this function calculates the polynom C[0] + C[1]*X^1 + C[2]*X^2 * C[3]*X^3 + C[4]*X^4 + C[5]*X^5 + C[6]*X^6 + C[7]*X^7

*)

F_POLY := ((((((( c[7] * x + c[6] ) * x + c[5] ) * x + c[4] ) * x + c[3] ) * x + c[2] ) * x + c[1] ) * x + c[0] ) ;


(* revision history
hm		20. may. 2008		rev 1.0
	original version

hm	18. mar. 2011	rev 1.1
	improved performance
*)

END_FUNCTION

// POUs/Mathematical/functions/F_POWER
FUNCTION F_POWER : REAL
VAR_INPUT
	a : REAL;
	x : REAL;
	n : REAL;
END_VAR


(*
version 1.0	1 sep 2006
programmer 	hugo
tested by		tobias

this function calculates the power equation f_power = a*x^n

*)

F_POWER := a * EXPT(X, N);

END_FUNCTION

// POUs/Mathematical/functions/F_QUAD
FUNCTION F_QUAD : REAL
VAR_INPUT
	X : REAL;
	A : REAL;
	B : REAL;
	C : REAL;
END_VAR


(*
version 1.1	18. Mar. 2011
programmer 	hugo
tested by		tobias

this function calculates the quadratic equation f_lin = a*x + b

*)

F_QUAD :=  (A * X + B) * X + C;

(* revision history

hm	1. sep. 2006	rev 1.0
	original version

hm	18. mar. 2001	rev 1.1
	improved performance
*)

END_FUNCTION

// POUs/Engineering/conversion/F_TO_C
FUNCTION F_TO_C : REAL
VAR_INPUT
	fahrenheit : REAL;
END_VAR


(*
version 1.1	11. mar. 2009
programmer 	hugo
tested BY		tobias

this FUNCTION converts fahrenheit TO celsius

*)

F_TO_C := (fahrenheit - 32.0) * 0.5555555555555;

(* revision history
hm	4. aug 2006	rev 1.0
	original version

hm	11. mar. 2009	rev 1.1
	real constants updated to new systax using dot

*)

END_FUNCTION

// POUs/Engineering/conversion/F_TO_OM
FUNCTION F_TO_OM : REAL
VAR_INPUT
	F : REAL;
END_VAR


(*
version 1.1	18. oct. 2008
programmer 	hugo
tested by	oscat

this function converts frequency to Omega F
Omega = 2*PI*F
*)

F_TO_OM := math.PI2 * F;


(* revision history
hm	22. jan. 2007	rev 1.0
	original version

hm	18. oct. 2008	rev 1.1
	unsing math constants

*)

END_FUNCTION

// POUs/Engineering/conversion/F_TO_PT
FUNCTION F_TO_PT : TIME
VAR_INPUT
	F : REAL;
END_VAR


(*
version 1.1	11. mar. 2009
programmer 	hugo
tested by		tobias

this function converts frequency to periode time  
*)

F_TO_PT := DWORD_TO_TIME(REAL_TO_DWORD(1.0 / F * 1000.0));


(* revision history

hm	4. aug. 2006	rev 1.0
	original version

hm	11. mar. 2009	rev 1.1
	real constants updated to new systax using dot

*)

END_FUNCTION

// POUs/Mathematical/FACT
FUNCTION FACT : DINT
VAR_INPUT
	X : INT;
END_VAR


(*
version 1.5	26. mar. 2011
programmer 	hugo
tested by		tobias

this function calculates the factorial of x

if the input is negative or higher then 12 the output will be -1.

*)

IF X >= 0 AND X <= 12 THEN
	FACT := math.FACTS[X];
ELSE
	FACT := -1;
END_IF;


(* working code without array
IF X > 12 OR X < 0 THEN
	FACT := -1;
ELSIF X < 7 THEN
	FACT := 1;
	FOR i := 2 TO X DO
		FACT := FACT * i;
	END_FOR;
ELSE
	FACT := 5040;
	FOR i := 8 TO X DO
		FACT := FACT * i;
	END_FOR;
END_IF;
*)

(* revision history
hm 4.3.2007		rev 1.1
	changed a critical error where while loop was indefinite.

hm	10.12.2007	rev 1.2
	start value for i has changed to 2 for better performance

hm	10. mar 2008	rev 1.3
	changed output of fact to dint to allow bigger values

hm	27. oct. 2008	rev 1.4
	optimized code

hm	26. mar. 2011	rev 1.5
	using array math.facts
*)

END_FUNCTION

// POUs/Engineering/signal processing/FADE
FUNCTION_BLOCK FADE
VAR_INPUT
	IN1 : REAL;
	IN2 : REAL;
	F : BOOL;
	TF : TIME;
	rst : BOOL;
END_VAR
VAR_OUTPUT
	Y : REAL;
END_VAR
VAR
	rmx : RMP_W;
END_VAR

(*
version 1.3	24. jan. 2009
programmer 	oscat
tested BY		oscat

FADE is used to crossfade between the inputs IN1 and IN2. The fade_over time is specified with TF.
When F = TRUE then Y = IN2 after the time TF, and when F = FALSE then Y = IN1.

*)

rmx(rst := rst AND NOT F, set := rst AND F, pt := TF, up := F);
Y := (in2 - In1) / 65535.0 * WORD_TO_REAL(rmx.out) + in1;


(* code for rev 1.1
IF rst THEN
	rmx(set := F, rst := NOT F);
ELSIF F AND (NOT rmx.high) THEN
	rmx(PT := TF, UP := TRUE, e := TRUE, rst := FALSE, set := FALSE);
ELSIF (NOT F) AND (NOT rmx.low) THEN
	rmx(PT := TF, UP := FALSE, e := TRUE, rst := FALSE, set := FALSE);
ELSE
	rmx(e := FALSE, rst := FALSE, set := FALSE);
END_IF;
Y := (WORD_TO_REAL(rmx.out) * in1 + WORD_TO_REAL(FF - rmx.out) * IN2) / FF;
*)


(* revision history
hm	26. dec 2007	rev 1.0
	original version

hm	18. oct. 2008	rev 1.1
	improved performance
	changed calls for rmp_w because rmp_w has chaged

hm	17. dec. 2008	rev 1.2
	function of input f was inverted

hm	24. jan. 2009	rev 1.3
	delted unused var FF
*)

END_FUNCTION_BLOCK

// POUs/Engineering/signal generators/RMP_W
FUNCTION_BLOCK RMP_W
VAR_INPUT
	SET : BOOL;
	PT : TIME;
	E : BOOL := TRUE;
	UP : BOOL := TRUE;
	RST : BOOL;
END_VAR
VAR_OUTPUT
	out : WORD;
	busy : BOOL;
	high : BOOL;
	low : BOOL;
END_VAR
VAR
	rmp : _RMP_W;
END_VAR

(*
version 2.0	23. oct. 2008
programmer 	oscat
tested BY	oscat

this ramp generator generates a Word wide ramp with 65535 steps
the generator has an asynchronous set and reset
the ramp is controlled by PT which is the total ramp time for a full sweep from 0..65535
an UD input controlls the direction Up or Down and the E input enables the ramp generation
a busy output indicates that the ramp is running, busy false means output is stable.
the outputs low and high will be true when the output has reached its max or min value.
*)

(* generate ramp *)
rmp(dir := UP, E := E, TR := PT, rmp := out);

(* set or reset operation *)
IF RST THEN
	out := 0;
ELSIF SET THEN
	out := 65535;
END_IF;

(* checks for outputs stable and reset or set busy flag *)
low := out = 0;
high := out = 65535;
busy := NOT (low OR high) AND E;


(* revision history:

hm 4.10.2006		rev 1.1
	added the busy output which signals that the ramp is running.

hm 22.1.2007		rev 1.2
	deleted unused variable step

hm	17.9.2007		rev 1.3
	replaced time() with t_plc_ms() for compatibility reasons

hm	28. sep 2007	rev 1.4
	added outputs on and off
	busy is now disabled while en is false
	new coding for higher accuracy and performance

hm	5. oct 2007	rev 1.5
	added statements to allow for PT to be t#0s output jumps to max or min immediately

hm	2. dec 2007	rev 1.6
	corrected an error in calculation of step response

hm	25. dec 2007	rev 1.7
	corrected an error while step response was too slow for fast rise times

hm	16. oct. 2008	rev 1.8
	improved performance

hm	18. oct. 2008	rev 1.9
	renamed inout EN to E for compatibility reasons

hm	23. oct. 2008	rev 2.0
	new code using _RMP_W
*)

END_FUNCTION_BLOCK

// POUs/Logic/FF edge triggered/FF_D2E
FUNCTION_BLOCK FF_D2E
VAR_INPUT
	D0 : BOOL;
	D1 : BOOL;
	CLK : BOOL;
	RST : BOOL;
END_VAR
VAR_OUTPUT
	Q0 : BOOL;
	Q1 : BOOL;
END_VAR
VAR
	edge : BOOL;
END_VAR

(*
version 1.3	14. mar. 2009
programmer 	hugo
tested by		oscat

dual D-type flip flop with reset and rising clock trigger

*)

IF rst THEN
	Q0 := FALSE;
	Q1 := FALSE;
ELSIF clk AND NOT edge THEN
	Q0 := D0;
	Q1 := D1;
END_IF;
edge := CLK;

(* revision history
hm	25. dec 2007	rev 1.0
	original version

hm	27. dec 2007	rev 1.1
	changed code for better performance

hm	30. oct. 200	rev 1.2
	deleted unnecessary init with 0

hm	14. mar. 2009	rev 1.3
	removed double assignments

*)

END_FUNCTION_BLOCK

// POUs/Logic/FF edge triggered/FF_D4E
FUNCTION_BLOCK FF_D4E
VAR_INPUT
	D0 : BOOL;
	D1 : BOOL;
	D2 : BOOL;
	D3 : BOOL;
	CLK : BOOL;
	RST : BOOL;
END_VAR
VAR_OUTPUT
	Q0 : BOOL;
	Q1 : BOOL;
	Q2 : BOOL;
	Q3 : BOOL;
END_VAR
VAR
	edge : BOOL;
END_VAR


(*
version 1.3	14. mar. 2009
programmer 	hugo
tested by		oscat

quad D-type flip flop with reset and rising clock trigger

*)

IF rst THEN
	Q0 := FALSE;
	Q1 := FALSE;
	Q2 := FALSE;
	Q3 := FALSE;
ELSIF clk AND NOT edge THEN
	Q0 := D0;
	Q1 := D1;
	Q2 := D2;
	Q3 := D3;
END_IF;
edge := CLK;

(* revision history
hm	4. aug 2006	rev 1.0
	original version

hm	27. dec 2007	rev 1.1
	changed code for better performance

hm	30. oct. 200	rev 1.2
	deleted unnecessary init with 0

hm	14. mar. 2009	rev 1.3
	removed double assignments

*)

END_FUNCTION_BLOCK

// POUs/Logic/FF edge triggered/FF_DRE
FUNCTION_BLOCK FF_DRE
VAR_INPUT
	SET : BOOL;
	D : BOOL;
	CLK : BOOL;
	RST : BOOL;
END_VAR
VAR_OUTPUT
	Q : BOOL;
END_VAR
VAR
	edge : BOOL;
END_VAR


(*
version 1.2	30. oct. 2008
programmer 	hugo
tested by	oscat

D-type flip flop with set, reset and rising clock trigger

*)

IF rst OR set THEN
	Q := NOT rst;
ELSIF clk AND NOT edge THEN
	Q := D;
END_IF;
edge := CLK;

(* revision history
hm	4. aug 2006		rev 1.0
	original version

hm	27. dec 2007	rev 1.1
	changed code for better performance

hm	30. oct. 2008	rev 1.2
	optimized performance
*)

END_FUNCTION_BLOCK

// POUs/Logic/FF edge triggered/FF_JKE
FUNCTION_BLOCK FF_JKE
VAR_INPUT
	SET : BOOL;
	J : BOOL;
	CLK : BOOL;
	K : BOOL;
	RST : BOOL;
END_VAR
VAR_OUTPUT
	Q : BOOL;
END_VAR
VAR
	edge : BOOL;
END_VAR


(*
version 1.2	30. oct. 2008
programmer 	hugo
tested by	oscat

JK-type flip flop with set, reset and rising clock trigger
set and reset are asynchron while the FF is rising edge triggered
J=0 and K=0 and CLK >>> no action
J=1 and K=0 and CLK >>> output = 1
J=0 and K=1 and CLK >>> output = 0
J=1 and K=1 and CLK >>> toggle output


*)

IF rst OR set THEN
	Q := NOT rst;
ELSIF clk AND NOT edge THEN
	IF J XOR K THEN Q := J;
	ELSE Q := K XOR Q;
	END_IF;
END_IF;
edge := CLK;

(* revision history
hm	4. aug 2006		rev 1.0
	original version

hm	27. dec 2007	rev 1.1
	changed code for better performance

hm	30. oct. 2008	rev 1.2
	optimized performance
*)

END_FUNCTION_BLOCK

// POUs/Logic/FF edge triggered/FF_RSE
FUNCTION_BLOCK FF_RSE
VAR_INPUT
	CS : BOOL;
	CR : BOOL;
	RST : BOOL;
END_VAR
VAR_OUTPUT
	Q : BOOL;
END_VAR
VAR
	es, er : BOOL;
END_VAR

(*
version 1.0	16. jul. 2008
programmer 	hugo
tested by	oscat

this is a rising edge triggered rs flip flop
a rising edge on CS sets Q = TRUE and a rising edge on CR sets Q = FALSE.
CR has priority over CS.

*)

IF rst THEN
	(* asynchronous reset *)
	Q := FALSE;
ELSIF CR AND NOT er THEN
	(* rising edge on CR *)
	Q := FALSE;
ELSIF CS AND NOT es THEN
	(* rising edge on CS *)
	Q := TRUE;
END_IF;

es := CS;
er := CR;

(* revision history

hm	16. jul. 2008	rev 1.0
	original version

*)

END_FUNCTION_BLOCK

// POUs/Mathematical/FIB
FUNCTION FIB : DINT
VAR_INPUT
	X : INT;
END_VAR
VAR
	t1, t2: DINT;
END_VAR

(*
version 1.3	26. mar. 2008
programmer 	hugo
tested by		tobias

this function calculates the fibonacci sequence

*)

IF X < 0 OR X > 46 THEN
	FIB := -1;
ELSIF x < 2 THEN
	FIB := X;
	RETURN;
ELSE
	(* the fibonacci number is the sum of the two suceeding fibonaci numbers *)
	(* we store the numbers alternatively in t1 and t2 depending on pt *)
	t2 := 1;
	WHILE X > 3 DO
		X := X-2;
		t1 := t1 + t2;
		t2 := t1 + t2;
	END_WHILE;
	IF X > 2 THEN t1 := t1 + t2; END_IF;
	fib := t1 + t2;
END_IF;

(* alternative code for very big numbers

IF X < 31 THEN
	fib := 0.4472136 * (expn(1.618034,X) - expn(-0.618034,X));
ELSE
	fib := 0.4472133 * expn(1.618034,X);
END_IF;

*)

(* revision history
hm		27. dec 2007	rev 1.0
	original version

hm		2. jan 2008	rev 1.1
	deleted unused variable pt

hm		10. mar 2008	rev 1.2
	changed output to dint instead of real

hm		26. mar. 2008	rev 1.3
	function now returns -1 for input < 0 or > 46

*)

END_FUNCTION

// POUs/Logic/memory/FIFO_16
FUNCTION_BLOCK FIFO_16
VAR_INPUT
	Din : DWORD;
	E : BOOL := TRUE;
	RD : BOOL;
	WD : BOOL;
	RST : BOOL;
END_VAR
VAR_OUTPUT
	Dout : DWORD;
	EMPTY : BOOL := TRUE;
	FULL : BOOL;
END_VAR
VAR
	fifo : ARRAY[0..n] OF DWORD;
	pr : INT;
	pw : INT;
END_VAR
VAR CONSTANT
	n : INT := 16;	(* changing this value will chage the number of stored elements in the fifo *)
END_VAR


(*
version 2.0	24. jul. 2009
programmer 	hugo
tested by		oscat

16 Dword FIFO memory
*)

IF RST THEN
	pw := pr;
	FULL := FALSE;
	EMPTY := TRUE;
	Dout := 0;
ELSIF E THEN
	IF NOT EMPTY AND RD THEN
		Dout := fifo[pr];
		pr := INC1(pr,n);
		EMPTY := pr = pw;
		FULL := FALSE;
	END_IF;
	IF NOT FULL AND WD THEN
		fifo[pw] := Din;
		pw := INC1(pw,n);
		FULL := pw = pr;
		EMPTY := FALSE;
	END_IF;
END_IF;


(* revision history

hm	4. aug. 2006	rev 1.0
	original version

hm	19. feb 2008	rev 1.1
	performance improvements

hm	17. oct. 2008	rev 1.2
	improved performance

ks	27. oct. 2008	rev 1.3
	optimized coding

hm	14. mar. 2009	rev 1.4
	removed double assignments

hm 24. jul. 2009	rev 2.0
	chaged inputs E and WR to E, WD and WR
	allow read and write in one cycle

*)

END_FUNCTION_BLOCK

// POUs/Logic/memory/FIFO_32
FUNCTION_BLOCK FIFO_32
VAR_INPUT
	Din : DWORD;
	E : BOOL := TRUE;
	RD : BOOL;
	WD : BOOL;
	RST : BOOL;
END_VAR
VAR_OUTPUT
	Dout : DWORD;
	EMPTY : BOOL := TRUE;
	FULL : BOOL;
END_VAR
VAR
	fifo : ARRAY[0..n] OF DWORD;
	pr : INT;
	pw : INT;
END_VAR
VAR CONSTANT
	n : INT := 32;	(* changing this value will chage the number of stored elements in the fifo *)
END_VAR

(*
version 2.0	24. jul. 2009
programmer 	hugo
tested by		oscat

32 Dword FIFO memory
*)

IF RST THEN
	pw := pr;
	FULL := FALSE;
	EMPTY := TRUE;
	Dout := 0;
ELSIF E THEN
	IF NOT EMPTY AND RD THEN
		Dout := fifo[pr];
		pr := INC1(pr,n);
		EMPTY := pr = pw;
		FULL := FALSE;
	END_IF;
	IF NOT FULL AND WD THEN
		fifo[pw] := Din;
		pw := INC1(pw,n);
		FULL := pw = pr;
		EMPTY := FALSE;
	END_IF;
END_IF;

(* revision history
hm	4. aug. 2006	rev 1.0
	original version

hm	19. feb 2008	rev 1.1
	performance improvements

hm	17. oct. 2008	rev 1.2
	improved performance

ks	27. oct. 2008 rev 1.3
	improved code

hm	14. mar. 2009	rev 1.4
	removed double assignments

hm 24. jul. 2009	rev 2.0
	chaged inputs E and WR to E, WD and WR
	allow read and write in one cycle

*)

END_FUNCTION_BLOCK

// POUs/Engineering/signal processing/FILTER_DW
FUNCTION_BLOCK FILTER_DW
VAR_INPUT
	X : DWORD;
	T : TIME;
END_VAR
VAR_OUTPUT
	Y : DWORD;
END_VAR
VAR
	last : DWORD;
	tx: DWORD;
	init: BOOL;
	Yi : REAL;
END_VAR

(*
version 1.1	3. nov. 2008
programmer 	hugo
tested by		oscat

FILTER_DW is an low pass filter with a programmable time T used for DWORD format.
 
*)

(* read system time *)
tx := T_PLC_MS();

(* startup initialisation *)
IF NOT init OR T = t#0s THEN
	init := TRUE;
	Yi := DWORD_TO_REAL(X);
ELSE
	Yi := Yi + (DWORD_TO_REAL(X) - DWORD_TO_REAL(Y)) * DWORD_TO_REAL(tx - last) / TIME_TO_REAL(T);
END_IF;
last := tx;

Y := REAL_TO_DWORD(Yi);



(*
hm 10. oct. 2008	rev 1.0
	original version

hm	3. nov. 2008	REV 1.1
	corrected an overflow problem
*)

END_FUNCTION_BLOCK

// POUs/Engineering/signal processing/FILTER_I
FUNCTION_BLOCK FILTER_I
VAR_INPUT
	X : INT;
	T : TIME;
END_VAR
VAR_OUTPUT
	Y : INT;
END_VAR
VAR
	Yi : DINT;
	last : DWORD;
	tx: DWORD;
	init: BOOL;
END_VAR

(*
version 1.0	8. nov. 2008
programmer 	hugo
tested by	oscat

FILTER_I is a low pass filter with a programmable time T used for INT format.
 
*)

(* read system time *)
tx := T_PLC_MS();

(* startup initialisation *)
IF NOT init OR T = t#0s THEN
	init := TRUE;
	Yi := INT_TO_DINT(X) * 1000;
ELSE
	(* to increase accuracy of the filter we calculate internal Yi wich is Y * 1000 *)
	Yi := Yi + INT_TO_DINT(X - Y) * DWORD_TO_DINT(tx - last) * 1000 / TIME_TO_DINT(T);
END_IF;
last := tx;
Y := DINT_TO_INT(yi / 1000);



(*
hm 8. nov. 2008	rev 1.0
	original version

*)

END_FUNCTION_BLOCK

// POUs/Engineering/signal processing/FILTER_MAV_DW
FUNCTION_BLOCK FILTER_MAV_DW
VAR_INPUT
	X : DWORD;
	N : UINT;
	RST : BOOL;
END_VAR
VAR_OUTPUT
	Y : DWORD;
END_VAR
VAR
	init: BOOL;
	buffer : ARRAY[0..31] OF DWORD;
	i: INT;
END_VAR
VAR_TEMP
	tmp: INT;
END_VAR

(*
version 1.3	23. feb. 2009
programmer 	hugo
tested by		oscat

FILTER_MAV_DW is a moving average filter with programmable length N for DWORD Data.
 
*)

(* limit N to size of buffer *)
N := MIN(N, 32);

(* startup initialisation *)
IF NOT init OR rst OR N = 0 THEN
	init := TRUE;
	tmp := UINT_TO_INT(N)-1;
	FOR i := 0 TO tmp DO
		buffer[i] := X;
	END_FOR;
	Y := X;
ELSE
	tmp := UINT_TO_INT(N);
	i := INC1(i, tmp);
	Y := Y + (X - buffer[i]) / N;
	buffer[i] := X;
END_IF;




(*
hm 13. oct. 2008	rev 1.0
	original version

hm	27. oct. 2008	rev 1.1
	added typecast to avoid warnings

hm	24. nov. 2008	rev 1.2
	added typecasts to avoid warnings
	avoid divide by 0 if N = 0

hm	23. feb. 2009	rev 1.3
	limit N to max array size

*)

END_FUNCTION_BLOCK

// POUs/Engineering/signal processing/FILTER_MAV_W
FUNCTION_BLOCK FILTER_MAV_W
VAR_INPUT
	X : WORD;
	N : UINT;
	RST : BOOL;
END_VAR
VAR_OUTPUT
	Y : WORD;
END_VAR
VAR
	init: BOOL;
	buffer : ARRAY[1..32] OF WORD;
	i: INT;
	sum : DWORD;
END_VAR
VAR_TEMP
	tmp : INT;
END_VAR

(*
version 1.4	26. MAR. 2011
programmer 	hugo
tested by		oscat

FILTER_MAV_W is a moving average filter with programmable length N for WORD Data.
 
*)

(* limit N to size of buffer *)
N := MIN(N, 32);

(* startup initialisation *)
IF NOT init OR rst OR N = 0 THEN
	init := TRUE;
	tmp := UINT_TO_INT(N) - 1;
	FOR i := 1 TO tmp DO
		buffer[i] := X;
	END_FOR;
	sum := Y * N;
	Y := X;
ELSE
	tmp := UINT_TO_INT(N);
	i := INC1(i, tmp);
	sum := sum + X - buffer[i];
	Y := DWORD_TO_WORD(sum / N);
	buffer[i] := X;
END_IF;



(*
hm 13. oct. 2008	rev 1.0
	original version

hm	18. oct. 2008	rev 1.1
	added typecast to avoid warnings

hm	24. nov. 2008	rev 1.2
	added typecasts to avoid warnings
	avoid devide by 0 if N = 0

hm	23. feb. 2009	rev 1.3
	limit N to max array size

hm	26. mar. 2011	rev 1.4
	corrected error in calculation
*)

END_FUNCTION_BLOCK

// POUs/Engineering/signal processing/FILTER_W
FUNCTION_BLOCK FILTER_W
VAR_INPUT
	X : WORD;
	T : TIME;
END_VAR
VAR_OUTPUT
	Y : WORD;
END_VAR
VAR
	last : DWORD;
	tx: DWORD;
	init: BOOL;
	tmp: DWORD;
END_VAR

(*
version 1.2	25. jan. 2011
programmer 	hugo
tested by	oscat

FILTER_W is an low pass filter with a programmable time T used for WORD format.
 
*)

(* read system time *)
tx := T_PLC_MS();

(* startup initialisation *)
IF NOT init OR T = T#0s THEN
	init := TRUE;
	last := tx;
	Y := X;
ELSIF Y = X THEN
	last := tx;
ELSE
	tmp :=  WORD_TO_DWORD(X - Y) * (tx - last) / TIME_TO_DWORD(T);
	IF tmp <> 0 THEN
		Y := DINT_TO_WORD(WORD_TO_DINT(Y) + DWORD_TO_DINT(tmp));
		last := tx;
	END_IF;
END_IF;

(*
hm 10. oct. 2008	rev 1.0
	original version

hm	3. nov. 2008	rev 1.1
	fixed overflow problem in formula

hm	25. jan. 2011	rev 1.2
	fixed error in formula
*)

END_FUNCTION_BLOCK

// POUs/Engineering/signal processing/FILTER_WAV
FUNCTION_BLOCK FILTER_WAV
VAR_INPUT
	X : REAL;
	W : ARRAY[0..15] OF REAL;
	RST : BOOL;
END_VAR
VAR_OUTPUT
	Y : REAL;
END_VAR
VAR
	init: BOOL;
	buffer : ARRAY[0..15] OF REAL;
	i: INT;
	n: INT;
END_VAR

(*
version 1.2	10. mar. 2009
programmer 	hugo
tested by		oscat

FILTER_WAV is a moving average filter with programmable length N for DWORD Data.

*)

(* startup initialisation *)
IF NOT init OR rst THEN
	init := TRUE;
	FOR i := 0 TO 15 DO
		buffer[i] := X;
	END_FOR;
	i := 15;
	Y := X;
ELSE
	i := INC1(i, 16);
	buffer[i] := X;
END_IF;

(* calculate the weighted average *)
Y := 0.0;
FOR n := 0 TO 15 DO
	Y := buffer[i] * W[n] + Y;
	i := DEC1(i, 16);
END_FOR;


(*
hm 	14. oct. 2008	rev 1.0
	original version

hm	27. oct. 2008	rev 1.1
	changed _DEC and _INC to DEC1 and INC1

hm	10. mar. 2009	rev 1.2
	real constants updated to new systax using dot

*)

END_FUNCTION_BLOCK

// POUs/String/FIND_CHAR
FUNCTION FIND_CHAR : INT
VAR_INPUT
	str : STRING(STRING_LENGTH);
	pos : INT;
END_VAR
VAR
	i: INT;
	pt : POINTER TO ARRAY[1..255] OF BYTE;
	stop: INT;
	X: BYTE;
END_VAR

(*
version 1.3	21. oct. 2008
programmer 	hugo
tested by	tobias

find_char searches str and returns the starting position of the first character that is not a control character.
control characters are the ascii character 00 .. 31 and 127

*)

pt := ADR(str);
stop := LEN(str);
FOR i := MAX(pos,1) TO stop DO;
	X := pt^[i];
	IF X > 31 AND ((setup.EXTENDED_ASCII AND X <> 127) OR (NOT setup.EXTENDED_ASCII AND X < 127)) THEN
		FIND_CHAR := i;
		RETURN;
	END_IF;
END_FOR;
FIND_CHAR := 0;


(* revision history
hm	29. feb 2008	rev 1.0
	original version

hm	26. mar. 2008	rev 1.1
	char will now accept extended ascii

hm	29. mar. 2008	rev 1.2
	changed STRING to STRING(STRING_LENGTH)

hm	21. oct. 2008	rev 1.3
	changes setup constants
	optimized code
*)

END_FUNCTION

// POUs/String/FIND_CTRL
FUNCTION FIND_CTRL : INT
VAR_INPUT
	str : STRING(STRING_LENGTH);
	pos : INT;
END_VAR
VAR
	i: INT;
	pt : POINTER TO ARRAY[1..255] OF BYTE;
	stop: INT;
	x: BYTE;
END_VAR

(*
version 1.2	29. mar. 2008
programmer 	hugo
tested by		tobias

find_ctrl searches str and returns the starting position of a control character
control characters are the ascii character 00 .. 31 and 127.

*)

pt := ADR(str);
stop := LEN(str);
FOR i := MAX(pos,1) TO stop DO;
	x := PT^[I];
	IF x < 32 OR X = 127 THEN
		FIND_CTRL := i;
		RETURN;
	END_IF;
END_FOR;
FIND_CTRL := 0;


(* revision history
hm	29. feb 2008	rev 1.0
	original version

hm	26. mar. 2008	rev 1.1
	character 127 is now recognized as control

hm	29. mar. 2008	rev 1.2
	changed STRING to STRING(STRING_LENGTH)
*)

END_FUNCTION

// POUs/String/FIND_NONUM
FUNCTION FIND_NONUM : INT
VAR_INPUT
	str : STRING(STRING_LENGTH);
	pos : INT;
END_VAR
VAR
	i: INT;
	pt : POINTER TO ARRAY[1..255] OF BYTE;
	end: INT;
	X: BYTE;
END_VAR

(*
version 1.3	21. oct. 2008
programmer 	hugo
tested by	tobias

find_noNum searches str and returns the first position which is not a number.
a number is characterized by a letter "0..9" or "."

*)

pt := ADR(str);
end := LEN(str);
FOR i := MAX(pos,1) TO end DO;
	X := pt^[i];
	IF (X < 48 AND X <> 46) OR X > 57 THEN
		FIND_NONUM := i;
		RETURN;
	END_IF;
END_FOR;
FIND_NONUM := 0;


(* revision history
hm	6. oct. 2006	rev 1.0
	original version

hm	29. feb 2008	rev 1.1
	added input pos to start search at position

hm	29. mar. 2008	rev 1.2
	changed STRING to STRING(STRING_LENGTH)

hm	21. oct. 2008	rev 1.3
	optimized code

*)

END_FUNCTION

// POUs/String/FIND_NUM
FUNCTION FIND_NUM : INT
VAR_INPUT
	str : STRING(STRING_LENGTH);
	pos : INT;
END_VAR
VAR
	i : INT;
	pt : POINTER TO ARRAY[1..255] OF BYTE;
	stop : INT;
	X: BYTE;
END_VAR

(*
version 1.2	29. mar. 2008
programmer 	hugo
tested by		tobias

find_Num searches str and returns the starting position of a number
a number is characterized by a letter "0..9" or "."

*)

pt := ADR(str);
stop := LEN(str);
FOR i := MAX(pos,1) TO stop DO;
	X := pt^[i];
	IF (X > 47 AND X < 58) OR X = 46 THEN
		FIND_NUM := i;
		RETURN;
	END_IF;
END_FOR;
FIND_NUM := 0;


(* revision history
hm	6. oct. 2006	rev 1.0
	original version

hm	29. feb 2008	rev 1.1
	added input pos to start search at position

hm	29. mar. 2008	rev 1.2
	changed STRING to STRING(STRING_LENGTH)

*)

END_FUNCTION

// POUs/String/FINDB
FUNCTION FINDB : INT
VAR_INPUT
	str1 : STRING(STRING_LENGTH);
	str2 : STRING(STRING_LENGTH);
END_VAR
VAR
	pos: INT;
	length: INT;
END_VAR

(*
version 1.3	29. mar. 2008
programmer 	hugo
tested by		tobias

the function find searches an str1 for the presence of str2 and returns the first position of str1 of the last presence in instring.
the function is similar to find except it searches from the right to left.
 a 0 is returned if the string is not found.

*)

length := LEN(str2);
FOR pos := LEN(str1) - length + 1 TO 1 BY -1 DO
	IF MID(str1,length,pos) = str2 THEN
		FindB := pos;
		RETURN;
	END_IF;
END_FOR;
FindB := 0;

(* revision history
hm	6. oct 2006		rev 1.0
	original version

hm	15 dec 2007		rev 1.1
	changed code for better performance

hm	29. feb 2008	rev 1.2
	added findb := 0 for compatibility reasons

hm	29. mar. 2008	rev 1.3
	changed STRING to STRING(STRING_LENGTH)
*)

END_FUNCTION

// POUs/String/FINDP
FUNCTION FINDP : INT
VAR_INPUT
	str : STRING(STRING_LENGTH);
	src : STRING(STRING_LENGTH);
	pos: INT;
END_VAR
VAR
	i: INT;
	ls: INT;
	lx: INT;
	stp: INT;
END_VAR

(*
version 1.2	29. mar. 2008
programmer 	hugo
tested by	tobias

the function findP searches a string str for the occurence of src beginning at the position pos.

*)

ls := LEN(str);
lx := LEN(src);
IF ls < lx OR lx = 0 THEN RETURN; END_IF;
stp := ls - lx + 1;
FOR i := MAX(pos,1) TO stp DO
	IF MID(str,lx,i) = src THEN
		FINDP := i;
		RETURN;
	END_IF;
END_FOR;
FINDP := 0;

(* revision histroy
hm	4. feb. 2008	rev 1.0
	original release

hm	29. feb 2008	rev 1.1
	ADDED MAX(pos,1) in loop initialization

hm	29. mar. 2008	rev 1.2
	changed STRING to STRING(STRING_LENGTH)
*)

END_FUNCTION

// POUs/String/FLOAT_TO_REAL
FUNCTION FLOAT_TO_REAL : REAL
VAR_INPUT
	FLT : STRING(20);
END_VAR
VAR
	pt : POINTER TO ARRAY[1..20] OF BYTE;
	i: INT;
	X: BYTE;
	sign: INT := 1;
	stop: INT;
	tmp: DINT;
	d : INT;
END_VAR

(*
version 1.3	23. oct. 2008
programmer 	hugo
tested by	oscat

FLOAT_TO_REAL converts a string to a REAL.
the function ignores all wrong characters.
the comma can be , or .
the exponent has to start with capital E or lowercase e .


*)

pt := ADR(FLT);
stop := LEN(FLT);

(* we first check for sign and exit if first number or dot is reached *)
FOR i := 1 TO stop DO
	X := pt^[i];
	IF X > 47 AND X < 58 OR X = 46 THEN
		EXIT;
	ELSIF X = 45 THEN
		(* code 45 is sign *)
		sign := -1;
	END_IF;
END_FOR;

(* now we scan numbers till end or dot or E is reached *)
FOR i := i TO stop DO
	X := pt^[i];
	IF X = 44 OR X = 46 OR X = 69 OR X = 101 THEN
		EXIT;
	(* calculate the value of the digit *)
	ELSIF X > 47 AND x < 58 THEN
		tmp := tmp * 10 + X - 48;
	END_IF;
END_FOR;

(* process the portion after the comma if comma or dot is reached exit if exponent starts *)
IF x = 44 OR X = 46 THEN
	FOR i := i + 1 TO stop DO
		X := pt^[i];
		IF X = 69 OR X = 101 THEN
			EXIT;
		ELSIF x > 47 AND x < 58 THEN
			tmp := tmp * 10 + X - 48;
			d := d - 1;
		END_IF;
	END_FOR;
END_IF;

(* process exponent if present *)
IF X = 69 OR X = 101 THEN
	d := d + DEC_TO_INT(RIGHT(FLT, stop - i));
END_IF;

FLOAT_TO_REAL :=  EXPN(10, d) * DINT_TO_REAL(TMP * SIGN);




(* revision histroy
hm	22. jun. 2008	rev 1.0
	original release

hm	2. oct. 2008	rev 1.1
	fixed an error, characters 8 and 9 would not be converted

hm	22. oct. 2008	rev 1.2
	last fix was not done correctly

hm	23. oct. 2008	rev 1.3
	optimzed code
*)

END_FUNCTION

// POUs/Engineering/automation/FLOW_CONTROL
 FUNCTION_BLOCK FLOW_CONTROL
VAR_INPUT
	IN : BOOL;
	REQ : BOOL;
	ENQ : BOOL;
	RST : BOOL;
END_VAR
VAR_INPUT CONSTANT
	T_AUTO : TIME := T#1h;
	T_DELAY : TIME := T#23h;
END_VAR
VAR_OUTPUT
	Q : BOOL;
	STATUS : BYTE;
END_VAR
VAR
	timer : TP_1D;
END_VAR


(*
version 1.0	28. jun. 2008
programmer 	hugo
tested by	oscat

FLOW_CONTROL switches a valves depending on the input in.
flow control also limits the maximum ontime of the valve and controls pressure on the output side.

*)

STATUS := 100;
IF RST THEN
	Q := FALSE;
	timer(rst := TRUE);
	timer.RST := FALSE;
	STATUS := 103;
ELSIF ENQ THEN
	IF IN THEN
		status := 101;
	END_IF;
	IF REQ THEN
		(* timer will generate a timed pulse after TP goes high *)
		timer.PT1 := T_AUTO;
		timer.PTD := T_DELAY;
		timer.IN := TRUE;
		STATUS := 102;
	END_IF;
END_IF;


(* set output and run timer *)
timer();
timer.IN := FALSE;
Q := (IN AND ENQ) OR timer.Q;



(* revision history
hm 	28. jun. 2008 	rev 1.0
	original version

*)

END_FUNCTION_BLOCK

// POUs/Logic/generators/TP_1D
FUNCTION_BLOCK TP_1D
VAR_INPUT
	IN : BOOL;
	PT1 : TIME;
	PTD : TIME;
	RST : BOOL;
END_VAR
VAR_OUTPUT
	Q : BOOL;
	W : BOOL;
END_VAR
VAR
	tx : TIME;
	start: TIME;
	ix: BOOL;
END_VAR


(*
version 1.0	28. jun. 2008
programmer 	hugo
tested by	oscat

TP_1D generates a pulse every time it is calles with in := TRUE.
the module will reset IN by itself so no clearing of in is necessary.
in addition the timer can be cleared asynchronously with rst.
also the rst input is cleared by the module itself.
the timer can be retriggered as often as necessary. it will count PT from the last trigger.
after the time PT1 is elapsed, the timer blocks itself for PT2 and only allow new sequences after PT2 has elapsed.


*)

(* read system timer *)
tx := DWORD_TO_TIME(T_PLC_MS());

IF RST THEN
	Q := FALSE;
	rst := FALSE;
	W := FALSE;
ELSIF W THEN
	IF tx - start >= PTD THEN
		W := FALSE;
	END_IF;
ELSIF IN AND NOT ix THEN
	Q := TRUE;
	start := tx;
	in := FALSE;
ELSIF tx - start >= PT1 THEN
	Q := FALSE;
	W := TRUE;
	start := tx;
END_IF;

ix := IN;



(* revision history
hm	28. jun. 2008
	original version

*)

END_FUNCTION_BLOCK

// POUs/Engineering/measurements/ONTIME
FUNCTION_BLOCK ONTIME
VAR_INPUT
	IN : BOOL;
	RST : BOOL;
END_VAR
VAR_IN_OUT
	SECONDS : UDINT;
	CYCLES : UDINT;
END_VAR
VAR
	tx: DWORD;
	last : DWORD;
	edge : BOOL;
	init: BOOL;
	ms: DWORD;
END_VAR

(*
version 2.5	18. mar. 2011
programmer 	oscat
tested by		tobias

ONTIME measures the ontime of a signal in seconds.
the output SECONDS is of type DWORD which results in a total measurement range of 1 second up to 136 years.
internally ontime works with a resolution of milliseconds

*)

(* read system time *)
tx := T_PLC_MS();

(* make sure the first cycle works correctly *)
IF NOT init THEN
	init := TRUE;
	last := tx;
	ms := 0;
END_IF;
IF RST THEN
	SECONDS := 0;
	CYCLES := 0;
	last := tx;
	ms := 0;
ELSIF IN THEN
	(* add the current milliseconds *)
	ms := (tx - last) + ms;
	IF ms >= 1000 THEN
		seconds := seconds + 1;
		ms := ms - 1000;
	END_IF;
	cycles := cycles + BOOL_TO_UINT(NOT edge);
END_IF;
last := tx;
edge := in;


(* revision history
hm 22.2.2007		rev 1.1
	changed VAR RETAIN PERSISTENT to VAR RETAIN for better compatibility
	wago lon contollers do not support persisitent

hm 2.8.2007		rev 1.2
	adding time up in a real number will automatically lead to the point where 
	small time scales like the cycle time will be below the resolution of real and therefore
	ontime would not increase in small steps as necessary
	the time is now measured internally in two  dwords and be converted to real only for
	output purposes.
	deleted the variable power because it was unnecessary

hm	16.9.2007		rev 1.3
	changes time() to T_plc_ms() for compatibility reasons

hm	2. dec. 2007	rev 1.4
	chaged code for better performance

hm	16. mar. 2008	rev 1.5
	added type conversions to avoid warnings under codesys 3.0

hm	21. oct. 2008	rev 2.0
	changed module for much better performance and allow for external result storage

hm	10. nov. 2008	rev 2.1
	increased internal resolution to milliseconds

hm	16. nov. 2008	rev 2.2
	changed typecast to avoid warnings

hm	17. dec. 2008	rev 2.3
	fixed an error when in would be true for more then 49 days

hm	17. jan 2011	rev 2.4
	init will not clear seconds and cycles, only rst clears these values	

hm	18. mar. 2011	rev 2.5
	reset was not working

*)

END_FUNCTION_BLOCK

// POUs/Engineering/conversion/PRESSURE
FUNCTION_BLOCK PRESSURE
VAR_INPUT
	mws : REAL;
	torr : REAL;
	att : REAL;
	atm : REAL;
	pa : REAL;
	bar : REAL;
END_VAR
VAR_OUTPUT
	Ymws : REAL;
	Ytorr : REAL;
	Yatt : REAL;
	Yatm : REAL;
	Ypa : REAL;
	Ybar : REAL;
END_VAR


(*
version 1.1	11. mar. 2009
programmer 	hugo
tested by		oscat

this function converts different pressure units
any unused input can simply be left open.
different inputs connected at the same time will be added up.
*)

Ybar := bar +
		pa * 1.0E-5 +
		0.980665 * att +
		1.01325 * atm +
		0.001333224 * torr +
		0.0980665 * mws;
Ymws := ybar * 10.1971621297793;
Ytorr := ybar * 750.0615050434140;
Yatt := ybar * 1.0197162129779;
yatm := ybar * 0.9869232667160;
Ypa := ybar * 100000.0;


(*
Druck, Pascal Pa 1 Pa = 1 N/m2 = 1 kg/(s2 E m) . 0,75 E 10.2 mmHg
mechanische 1 MPa = 1 N/mm2 . fur Festigkeitsangaben
Spannung Bar bar 1 bar = 105 Pa = 103 mbar = 105 kg/(s2 E m)
Millimeter- mmHg 1 mmHg = 133,322 Pa = 1,333 22 mbar
Quecksilbersaule . nur in Heilkunde zulassig
physik. Atmosphare atm 1 atm = 1,013 25 bar
techn. Atmosphare at 1 at = 1 kp/cm2 = 0,980665 bar
Torr Torr 1 Torr = (101325/760) Pa = 1,333224 mbar
Meter-Wassersaule mWS 1 mWS = 9806,65 Pa = 98,0665 mbar
psi lbf/in2 1 lbf/in2 = 68,947 57 mbar = 6894,757 Pa

*)

(* revision history

hm	27. mar. 2007	rev 1.0
	original version

hm	11. mar. 2009	rev 1.1
	improved code

*)

END_FUNCTION_BLOCK

// POUs/Engineering/measurements/FLOW_METER
FUNCTION_BLOCK FLOW_METER
VAR_INPUT
	VX : REAL;
	E : BOOL;
	RST : BOOL;
END_VAR
VAR_INPUT CONSTANT
	PULSE_MODE : BOOL;
	UPDATE_TIME : TIME := t#1s;
END_VAR
VAR_OUTPUT
	F : REAL;
END_VAR
VAR_IN_OUT
	X : REAL;
	Y : UDINT;
END_VAR
VAR
	tx, tl : TIME;
	int1 : INTEGRATE;
	init: BOOL;
	e_last : BOOL;
	tmp: INT;
	x_last : REAL;
	y_last : UDINT;
END_VAR

(*
version 1.0	23. jan. 2011
programmer 	hugo
tested by	oscat

Flow meter measures flow according to gated time or pulses.

*)

IF NOT init THEN	(* init on power up *)
	init := TRUE;
	tl := tx;
	x_last := X;
	y_last := Y;
	int1.K := 2.7777777777777777E-4;
END_IF;

(* run integrator *)
int1(E := NOT (RST OR PULSE_MODE) AND E, X := VX, Y := X);	(* gated operation *)

IF RST THEN		(* reset *)
	X := 0.0;
	Y := 0;
	tl := tx;
	x_last := 0.0;
	y_last := 0;
ELSIF E AND PULSE_MODE THEN	(* check for pulse mode *)
	IF NOT e_last THEN X := X + VX; END_IF;
END_IF;
e_last := E;

(* reduce X to be less than 1 and increase Y respectively *)
IF X > 1.0 THEN
	tmp := FLOOR(X);
	Y := Y + INT_TO_UDINT(tmp);
	X := X - INT_TO_REAL(tmp);
END_IF;

(* calculate the current flow *)
tx := DWORD_TO_TIME(T_PLC_MS());
IF tx - tl >= UPDATE_TIME AND UPDATE_TIME > t#0s THEN
	F := (UDINT_TO_REAL(Y - y_last) + X - x_last) / TIME_TO_REAL(tx - tl) * 3.6E6;
	y_last := Y;
	x_last := X;
	tl := tx;
END_IF;



(* revision history
hm	23. jan. 2011	rev 1.0
	original version

*)

END_FUNCTION_BLOCK

// POUs/String/FSTRING_TO_BYTE
FUNCTION FSTRING_TO_BYTE : BYTE
VAR_INPUT
	IN : STRING(12);
END_VAR


(*
version 1.1	20. sep. 2008
programmer 	hugo
tested by		oscat

FSTRING_TO_BYTE converts a formatted string into a byte.
the string can be of the form 2#01010, 8#7234, 16#2AD3 and 1234

*)

IF LEFT(IN, 2) = '2#' THEN
	(* we need to convert binary *)
	FSTRING_TO_BYTE := BIN_TO_BYTE(RIGHT(in, LEN(in) - 2));
ELSIF LEFT(in, 2) = '8#' THEN
	(* weneed to convert octals *)
	FSTRING_TO_BYTE := OCT_TO_BYTE(RIGHT(in, LEN(in) - 2));
ELSIF LEFT(in, 3) = '16#' THEN
	(* we need to convert hexadecimal *)
	FSTRING_TO_BYTE := HEX_TO_BYTE(RIGHT(in, LEN(in) - 3));
ELSE
	(* we assume decimal representation *)
	FSTRING_TO_BYTE := DEC_TO_BYTE(CLEAN(in,'0123456789'));
END_IF;


(* revision histroy
hm	18. jun. 2008	rev 1.0
	original release

hm	20. sep. 2008	rev 1.1
	changed length of input string from 20 to 12
*)

END_FUNCTION

// POUs/String/OCT_TO_BYTE
FUNCTION OCT_TO_BYTE : BYTE
VAR_INPUT
	OCT : STRING(10);
END_VAR
VAR
	pt : POINTER TO BYTE;
	i: INT;
	X: BYTE;
	stop: INT;
END_VAR

(*
version 1.1	20. sep. 2008
programmer 	hugo
tested by		oscat

OCT_TO_BYTE converts a octagonal string into a byte.

*)

pt := ADR(oct);
stop := LEN(oct);
FOR I := 1 TO stop DO
	(* read the first character and subtract 48 to get value in decimal 0 = 48 *)
	x := pt^;
	(* calculate the value of the digit *)
	IF X > 47 AND x < 56 THEN
		OCT_TO_BYTE := SHL(OCT_TO_BYTE,3) + X - 48;
	END_IF;
	pt := pt + 1;
END_FOR;



(* revision histroy
hm	18. jun. 2008	rev 1.0
	original release

hm	20. sep. 2008	rev 1.1
	changed length of input string from 20 to 10

*)

END_FUNCTION

// POUs/String/HEX_TO_BYTE
FUNCTION HEX_TO_BYTE : BYTE
VAR_INPUT
	HEX : STRING(5);
END_VAR
VAR
	pt : POINTER TO BYTE;
	i: INT;
	X: BYTE;
	stop: INT;
END_VAR

(*
version 1.1	20. sep. 2008
programmer 	hugo
tested by		oscat

HEX_TO_BYTE converts a Hexadecimal string into a byte.

*)

pt := ADR(hex);
stop := LEN(hex);
FOR I := 1 TO stop DO
	(* read the first character and subtract 48 to get value in decimal 0 = 48 *)
	x := pt^;
	(* calculate the value of the digit *)
	IF X > 47 AND x < 58 THEN
		HEX_TO_BYTE := SHL(HEX_TO_BYTE,4) + X - 48;
	ELSIF X > 64 AND X < 71 THEN
		HEX_TO_BYTE := SHL(HEX_TO_BYTE,4) + X - 55;
	ELSIF X > 96 AND X < 103 THEN
		HEX_TO_BYTE := SHL(HEX_TO_BYTE,4) + X - 87;
	END_IF;
	pt := pt + 1;
END_FOR;




(* revision histroy
hm	18. jun. 2008	rev 1.0
	original release

hm	20. sep.2008	rev 1.1
	changed length of input string from 20 to 5

*)

END_FUNCTION

// POUs/String/FSTRING_TO_DT
FUNCTION FSTRING_TO_DT : DT
VAR_INPUT
	SDT : STRING(60);
	FMT : STRING(60);
END_VAR
VAR CONSTANT
	ignore: STRING(1) := '*';  (* ignore character is * *)
	fchar : STRING(1) := '#';  (* format character is # *)
END_VAR
VAR
	c: STRING(1);
	tmp: STRING(20);
	end: INT;
	dy : INT := 1970;
	dm : INT := 1;
	dd : INT := 1;
	th : INT;
	tm : INT;
	ts : INT;
END_VAR


(*
version 1.0	24. sep. 2008
programmer 	hugo
tested by	oscat

FSTRING_TO_DT converts Formatted String into a DT value.

*)

(* scan input string *)
WHILE fmt <> '' DO
	c := LEFT(fmt,1);
	IF c = ignore THEN
		(* skip ignore characters *)
		fmt := DELETE(fmt,1,1);
		sdt := DELETE(sdt,1,1);
	ELSIF C = fchar THEN
		(* format chracter found skip format char and read identifier *)
		(* store format identifier in c and skip to next char in fmt *)
		c := MID(fmt,1,2);
		fmt := DELETE(fmt,2,1);
		(* extract the substring until the end of sdt or to next char of fmt *)
		IF fmt = '' THEN
			tmp := sdt;
		ELSE
			(* serach for end of substring *)
			end := FIND(sdt, LEFT(fmt,1))-1;
			tmp := LEFT(sdt, end);
			sdt := DELETE(sdt, end,1);
		END_IF;
		(* extract information from substring *)
		IF c = 'Y' THEN
			dy := STRING_TO_INT(tmp);
			IF dy < 100 THEN dy := dy + 2000; END_IF;
		ELSIF c = 'M' THEN
			dm := STRING_TO_INT(tmp);
		ELSIF c = 'N' THEN
			dm := FSTRING_TO_MONTH(tmp,0);
		ELSIF c = 'D' THEN
			dd := STRING_TO_INT(tmp);
		ELSIF c = 'h' THEN
			th := STRING_TO_INT(tmp);
		ELSIF c = 'm' THEN
			tm := STRING_TO_INT(tmp);
		ELSIF c = 's' THEN
			ts := STRING_TO_INT(tmp);
		END_IF;
	ELSIF c = LEFT(sdt,1) THEN
		(* skip matching characters *)
		fmt := DELETE(fmt,1,1);
		sdt := DELETE(sdt,1,1);
	ELSE
		RETURN;
	END_IF;
END_WHILE;

FSTRING_TO_DT := SET_DT(dy,dm,dd,th,tm,ts);


(* revision histroy
hm	24. sep. 2008	rev 1.0
	original release


*)

END_FUNCTION

// POUs/String/FSTRING_TO_MONTH
FUNCTION FSTRING_TO_MONTH : INT
VAR_INPUT
	MTH : STRING(20);
	LANG : INT;
END_VAR
VAR
	lx: INT;
END_VAR


(*
version 1.2	25. oct 2008
programmer 	hugo
tested by	oscat

FSTRING_TO_MONTH converts a string into a month, the string can be a name for the month or a number.
the function is language sensitve when LANG > 1 and checks for all languages when LANG = 0

*)

IF LANG = 0 THEN lx := LANGUAGE.DEFAULT; ELSE lx := MIN(LANG, LANGUAGE.LMAX); END_IF;
MTH := TRIM(mth);
MTH := CAPITALIZE(LOWERCASE(MTH));

FOR FSTRING_TO_MONTH := 1 TO 12 DO
	IF MTH = language.MONTHS[lx, FSTRING_TO_MONTH] THEN RETURN; END_IF;
	IF MTH = language.MONTHS3[lx, FSTRING_TO_MONTH] THEN RETURN; END_IF;
END_FOR;

(* since no name matched try to decode as integer *)
FSTRING_TO_MONTH := STRING_TO_INT(MTH);




(* revision histroy
hm	25. sep. 2008	rev 1.0
	original release

hm	19. oct. 2008	rev 1.1
	changed language setup constants

hm	25. oct. 2008	rev 1.2
	optimized code
*)

END_FUNCTION

// POUs/String/FSTRING_TO_DWORD
FUNCTION FSTRING_TO_DWORD : DWORD
VAR_INPUT
	IN : STRING(40);
END_VAR


(*
version 1.1	20. sep. 2008
programmer 	hugo
tested by		oscat

FSTRING_TO_BYTE converts a formatted string into a byte.
the string can be of the form 2#01010, 8#7234, 16#2AD3 and 1234

*)

IF LEFT(IN, 2) = '2#' THEN
	(* we need to convert binary *)
	FSTRING_TO_DWORD := BIN_TO_DWORD(RIGHT(in, LEN(in) - 2));
ELSIF LEFT(in, 2) = '8#' THEN
	(* weneed to convert octals *)
	FSTRING_TO_DWORD := OCT_TO_DWORD(RIGHT(in, LEN(in) - 2));
ELSIF LEFT(in, 3) = '16#' THEN
	(* we need to convert hexadecimal *)
	FSTRING_TO_DWORD := HEX_TO_DWORD(RIGHT(in, LEN(in) - 3));
ELSE
	(* we assume decimal representation *)
	FSTRING_TO_DWORD := DEC_TO_DWORD(CLEAN(in,'0123456789'));
END_IF;


(* revision histroy
hm	18. jun. 2008	rev 1.0
	original release

hm	20. sep. 2008	rev 1.1
	changed length of input dtring from 20 to 40


*)

END_FUNCTION

// POUs/String/OCT_TO_DWORD
FUNCTION OCT_TO_DWORD : DWORD
VAR_INPUT
	OCT : STRING(20);
END_VAR
VAR
	pt : POINTER TO BYTE;
	i: INT;
	X: BYTE;
	stop: INT;
END_VAR

(*
version 1.0	18. jun 2008
programmer 	hugo
tested by	oscat

OCT_TO_DWORD converts a octagonal string into a dword.

*)

pt := ADR(oct);
stop := LEN(oct);
FOR I := 1 TO stop DO
	(* read the first character and subtract 48 to get value in decimal 0 = 48 *)
	x := pt^;
	(* calculate the value of the digit *)
	IF X > 47 AND x < 56 THEN
		OCT_TO_DWORD := SHL(OCT_TO_DWORD,3) + X - 48;
	END_IF;
	pt := pt + 1;
END_FOR;




(* revision histroy
hm	18. jun. 2008	rev 1.0
	original release


*)

END_FUNCTION

// POUs/String/HEX_TO_DWORD
FUNCTION HEX_TO_DWORD : DWORD
VAR_INPUT
	Hex : STRING(20);
END_VAR
VAR
	pt : POINTER TO BYTE;
	i: INT;
	X: BYTE;
	stop: INT;
END_VAR

(*
version 1.4	18. jun. 2008
programmer 	hugo
tested by	tobias

HEX_TO_DWORD converts a Hexadecimal string into a DWORD.

*)

pt := ADR(hex);
stop := LEN(hex);
FOR I := 1 TO stop DO
	(* read the first character and subtract 48 to get value in decimal 0 = 48 *)
	x := pt^;
	(* calculate the value of the digit *)
	IF X > 47 AND x < 58 THEN
		HEX_TO_DWORD := SHL(HEX_TO_DWORD,4) + X - 48;
	ELSIF X > 64 AND X < 71 THEN
		HEX_TO_DWORD := SHL(HEX_TO_DWORD,4) + X - 55;
	ELSIF X > 96 AND X < 103 THEN
		HEX_TO_DWORD := SHL(HEX_TO_DWORD,4) + X - 87;
	END_IF;
	pt := pt + 1;
END_FOR;



(* revision histroy
hm	2.10.2007		rev 1.0
	original release

hm	19.11.2007		rev 1.1
	changed type of function from int to dword

hm 	4. mar 2008		rev 1.2
	added support for a..f and return 0 for invalid string

hm	29. mar. 2008	rev 1.3
	changed STRING to STRING(8)

hm	18. jun. 2008	rev 1.4
	changed input hex to STRING(20)
	function now ignores wrong characters
*)

END_FUNCTION

// POUs/String/FSTRING_TO_WEEK
FUNCTION FSTRING_TO_WEEK : BYTE
VAR_INPUT
	WEEK : STRING(60);
	LANG : INT;
END_VAR
VAR
	pos: INT;
END_VAR


(*
version 1.1	25. oct. 2008
programmer 	hugo
tested by	oscat

FSTRING_TO_WEEK converts a list of weekdays into a byte where each bit represents a day of the week.
bit 6 = mo, 0 = su;

*)

pos := FIND(WEEK, ',');
WHILE pos > 0 DO
	FSTRING_TO_WEEK := FSTRING_TO_WEEK OR SHR(BYTE#128, FSTRING_TO_WEEKDAY(MID(WEEK, pos - 1, 1), LANG));
	WEEK := RIGHT(WEEK, LEN(Week) - pos);
	pos := FIND(WEEK, ',');
END_WHILE;
FSTRING_TO_WEEK := (FSTRING_TO_WEEK OR SHR(BYTE#128, FSTRING_TO_WEEKDAY(WEEK, LANG))) AND BYTE#127;


(* revision histroy
hm	18. jun. 2008	rev 1.0
	original release

hm	25. oct. 2008	rev 1.1
	using language defauls and input lang
*)

END_FUNCTION

// POUs/String/FSTRING_TO_WEEKDAY
FUNCTION FSTRING_TO_WEEKDAY : INT
VAR_INPUT
	WDAY : STRING(20);
	LANG : INT;
END_VAR
VAR
	tmp: STRING(2);
	i: INT;
	ly: INT;
END_VAR


(*
version 1.2	25. oct. 2008
programmer 	hugo
tested by	oscat

FSTRING_TO_WEEKDAY converts a weekday string into an integer 1..7.

*)

IF LANG = 0 THEN ly := LANGUAGE.DEFAULT; ELSE ly := MIN(LANG, LANGUAGE.LMAX); END_IF;
(* tmp needs to be calculated first otherwise find can return wrong values *)
tmp := TRIM(wday);
tmp := CAPITALIZE(LOWERCASE(tmp));
FOR i := 1 TO 7 DO
	IF language.WEEKDAYS2[ly, i] = tmp THEN
		FSTRING_TO_WEEKDAY := i;
		RETURN;
	END_IF;
END_FOR;
FSTRING_TO_WEEKDAY := STRING_TO_INT(WDAY);




(* revision histroy
hm	18. jun. 2008	rev 1.0
	original release

hm	18. jul. 2008	rev 1.1
	changed nested call of left(trim()) for compatibility reasons

hm	25. oct. 2008	rev 1.2
	using language constants
*)

END_FUNCTION

// POUs/Mathematical/functions/FT_AVG
FUNCTION_BLOCK FT_AVG
VAR_INPUT
	IN : REAL;
	E : BOOL := TRUE;
	N : INT := 32;
	RST : BOOL;
END_VAR
VAR_OUTPUT
	AVG : REAL;
END_VAR
VAR
	buff : DELAY;
	i: INT;
	init : BOOL;
END_VAR

(*
version 1.5	10. mar. 2009
programmer 	hugo
tested by		oscat

this function calculates the moving average over n samples from a sequential input
the input values are shifted into an N deep buffer and the avg of this buffer is diplayed at anytime on the output.
a rst will load the buffer with the current in value..

*)

(* limit n to a max of 32 because delay can do max 32 cycles *)
buff.N := LIMIT(0, N, 32);

IF NOT init OR rst THEN
	FOR i := 1 TO N DO
		buff(in := in);
	END_FOR;
	avg := in;
	init := TRUE;
ELSIF E THEN
	buff(in := in);
	avg := avg + (in - buff.out ) / INT_TO_REAL(N);
END_IF;

(* revision history

hm	7. jan. 2007	rev 1.1
	chaged rst logic to load the buffer with the actual input value instead of 0.
	added en input to allow better control of signal flow
	added init to load the buffer with in at startup to avoid rampup at beginning.
	deleted unused variable cnt.

hm	14. jun. 2008	rev 1.2
	set default for input en = TRUE and N = 32

hm	10. oct. 2008	rev 1.3
	improved performance

hm	18. oct. 2008	rev 1.4
	changed input en to e for compatibility reasons

hm	10. mar. 2009	rev 1.5
	added type conversion for compatibility reasons

*)

END_FUNCTION_BLOCK

// POUs/Engineering/control/FT_IMP
FUNCTION_BLOCK FT_IMP
VAR_INPUT
	in : REAL;
	T : TIME;
	K : REAL := 1.0;
END_VAR
VAR_OUTPUT
	out : REAL;
END_VAR
VAR
	t1 : FT_PT1;
END_VAR

(*
version 1.1	3 Jan 2007
programmer 	hugo
tested by	oscat

FT_IMP is 	an impulse filter (high pass filter) with the time T and factor K.
 
*)

T1(in:= in, T:=T);
out := (in - t1.out) * K;

(*
hm 3.1.2007	rev 1.1
	added factor K

*)

END_FUNCTION_BLOCK

// POUs/Engineering/control/FT_INT2
FUNCTION_BLOCK FT_INT2
VAR_INPUT
	IN : REAL;
	K : REAL := 1.0;
	RUN : BOOL := TRUE;
	RST : BOOL;
	OUT_MIN : REAL := -1.0E38;
	OUT_MAX : REAL := 1.0E38;
END_VAR
VAR_OUTPUT
	OUT : REAL;
	LIM : BOOL;
END_VAR
VAR
	integ: INTEGRATE;
	ix : REAL;
	val : REAL2;
END_VAR


(*
version 1.2	11. mar. 2009
programmer 	hugo
tested by		oscat

FT_int2 is an integrator with input IN and factor K.
integration is only done while run = true, if run is false integration is stopped and the out remains at the last value.
if run is left unconnected, run is considered true by the function block.
the out_min and out_max values can be set to ,imit the output value range. 
the default for K is 1.
FT_INT2 has double presision accuracy (14 digits).


*)

IF RST THEN
	val := R2_SET(0.0);
	out := 0.0;
ELSE
	integ(X := IN, E := RUN, K := K, Y := ix);
	val := R2_ADD(val, ix);
	ix := 0.0;
	OUT := val.RX;
END_IF;

(* check output for limits *)
IF out > OUT_MIN AND out < OUT_MAX THEN
	LIM := FALSE;
ELSE
	OUT := LIMIT(OUT_MIN, OUT, OUT_MAX);
	val := R2_SET(OUT);
	LIM := TRUE;
END_IF;



(*	revision history
hm	2. jun. 2008	rev 1.0
	original version

hm	5. nov. 2008	rev 1.1
	rewritten code using integrate

hm	11. mar. 2009	rev 1.2
	real constants updated to new systax using dot

*)

END_FUNCTION_BLOCK

// POUs/Mathematical/Double Precision/R2_SET
FUNCTION R2_SET : REAL2
VAR_INPUT
	X : REAL;
END_VAR


(*
version 1.1	10. mar. 2009
programmer 	hugo
tested by		tobias

R2_set sets a double precision real to a single real value.

*)

R2_SET.RX := X;
R2_SET.R1 := 0.0;


(* revision history
hm	2. jun. 2008	rev 1.0
	original version

hm	10. mar. 2009	rev 1.1
	real constants updated to new systax using dot

*)

END_FUNCTION

// POUs/Mathematical/functions/FT_MIN_MAX
FUNCTION_BLOCK FT_MIN_MAX
VAR_INPUT
	in : REAL;
	rst : BOOL;
END_VAR
VAR_OUTPUT
	mx : REAL;
	mn : REAL;
END_VAR
VAR
	init: BOOL;
END_VAR

(*
version 1.0	1 sep 2006
programmer 	hugo
tested by		tobias

this function block stores the min and max value of an input signal.
when rst is true the mn and mx outputs are set to the in value.
when a rst is never active the function autoresets to the in value at startup.
since the input might not be present at first cycle the mn and mx are set during second cycle.

*)

IF rst OR NOT init THEN
	mn := in;
	mx := in;
	init := TRUE;
ELSIF in < mn THEN mn := in;
ELSIF in > mx THEN mx := in;
END_IF;

END_FUNCTION_BLOCK

// POUs/Engineering/control/FT_PD
FUNCTION_BLOCK FT_PD
VAR_INPUT
	IN : REAL;
	KP : REAL := 1.0;
	TV : REAL := 1.0;
END_VAR
VAR_OUTPUT
	Y : REAL;
END_VAR
VAR
	diff : FT_DERIV;
END_VAR

(*
version 1.0	3. jun 2008
programmer 	hugo
tested by		tobias

FT_PD is a PD controller.
The PD controller works according to the fomula Y = KP *(IN + DERIV(e) ).

*)

(* run differentiator *)
diff(IN := IN, K := TV);

(* combine both values *)
Y := KP * (diff.out + IN);



(* revision history
hm 	3. jun. 2008 	rev 1.0
	original version


*)

END_FUNCTION_BLOCK

// POUs/Engineering/control/FT_PDT1
FUNCTION_BLOCK FT_PDT1
VAR_INPUT
	IN : REAL;
	KP : REAL := 1.0;
	TV : REAL := 1.0;
	T1 : REAL := 1.0;
END_VAR
VAR_OUTPUT
	Y : REAL;
END_VAR
VAR
	diff : FT_DERIV;
	TP : FT_PT1;
END_VAR

(*
version 1.0	3. jun 2008
programmer 	hugo
tested by		tobias

FT_PD is a PD controller.
The PD controller works according to the fomula Y = KP *(IN + DERIV(e) ).

*)

(* run differentiator *)
diff(IN := IN, K := TV);

(* Run PT1 filter *)
tp(in := diff.out, T := REAL_TO_TIME(T1));

(* combine both values *)
Y := KP * (tp.out + IN);



(* revision history
hm 	3. jun. 2008 	rev 1.0
	original version


*)

END_FUNCTION_BLOCK

// POUs/Engineering/control/FT_PID
FUNCTION_BLOCK FT_PID
VAR_INPUT
	IN : REAL;
	KP : REAL := 1.0;
	TN : REAL := 1.0;
	TV : REAL := 1.0;
	ILIM_L : REAL := -1.0E38;
	ILIM_H : REAL := 1.0E38;
	IEN : BOOL := TRUE;
	RST : BOOL;
END_VAR
VAR_OUTPUT
	Y : REAL;
	LIM : BOOL;
END_VAR
VAR
	integ : FT_INT;
	diff : FT_DERIV;
END_VAR

(*
version 2.1	11. mar. 2009
programmer 	hugo
tested by		tobias

FT_PI is a PI controller.
The PID controller works according to the fomula Y = IN *(KP+ KI * INTEG(e) ).
a rst will reset the integrator to 0
ilim_h and iLim_l set the possible output range of the internal integrator.
the output flags lim will signal that the output limits are active.

default values for KP = 1, KI = 1, ILIM_L = -1E37, iLIM_H = +1E38.
*)

(* run integrator only if TN > 0 *)
IF TN > 0.0 THEN
	integ(IN := IN, K := 1.0 / TN, RUN := IEN, RST := RST, OUT_MIN := ILIM_L, OUT_MAX := ILIM_H);
ELSE
	integ(RST := FALSE);
END_IF;

(* run differentiator *)
diff(IN := IN, K := TV);

(* combine both values *)
Y := KP * (integ.Out + diff.out + IN);

(* check if integrator has reached its limits and set overflow *)
LIM := integ.LIM;



(* revision history
hm 3. jun. 2008 	rev 2.0
	original version

hm	11. mar. 2009	rev 2.1
	real constants updated to new systax using dot

*)

END_FUNCTION_BLOCK

// POUs/Engineering/control/FT_PIDW
FUNCTION_BLOCK FT_PIDW
VAR_INPUT
	IN : REAL;
	KP : REAL := 1.0;
	TN : REAL := 1.0;
	TV : REAL := 1.0;
	LIM_L : REAL := -1.0E38;
	LIM_H : REAL := 1.0E38;
	RST : BOOL;
END_VAR
VAR_OUTPUT
	Y : REAL;
	LIM : BOOL;
END_VAR
VAR
	integ : INTEGRATE;
	diff : FT_DERIV;
	YI: REAL;
END_VAR

(*
version 1.2	11. mar. 2009
programmer 	hugo
tested by		oscat

FT_PIDW is a PID controller with dynamic wind_up reset.
The PID controller works according to the fomula Y = KP *(IN + KI * INTEG(e) + DERIV(e) ).
a rst will reset the integrator to 0
lim_h and Lim_l set the possible output range of the internal integrator.
the output flags lim will signal that the output limits are active.

default values for KP = 1, KI = 1, ILIM_L = -1E37, iLIM_H = +1E38.
*)

(* run the integrator *)
IF tn = 0.0 OR rst THEN
	integ(E := FALSE, Y := YI);
	YI := 0.0;
ELSE
	integ(X := IN, K := 1.0 / TN, E := NOT LIM, Y := YI);
END_IF;

(* add up integrator and linear part *)
Y := KP * (IN + YI);

(* run differentiator *)
diff(IN := IN, K := TV);

(* set lim before differentiator is added to stop integrator if necessary *)
IF Y > LIM_L AND Y < LIM_H THEN
	LIM := FALSE;
ELSE
	LIM := TRUE;
END_IF;

(* add differential part and limit output Y *)

Y := LIMIT(LIM_L, Y + KP * diff.out, LIM_H);




(* revision history
hm 3. jun. 2008 	rev 1.0
	original version

hm	5. nov. 2008	rev 1.1
	changed code to use integrate

hm	11. mar. 2009	rev 1.2
	real constants updated to new systax using dot

*)

END_FUNCTION_BLOCK

// POUs/Engineering/control/FT_PIW
FUNCTION_BLOCK FT_PIW
VAR_INPUT
	IN : REAL;
	KP : REAL := 1.0;
	KI : REAL := 1.0;
	LIM_L : REAL := -1E38;
	LIM_H : REAL := 1E38;
	RST : BOOL;
END_VAR
VAR_OUTPUT
	Y : REAL;
	LIM : BOOL;
END_VAR
VAR
	integ : FT_INT;
END_VAR

(*
version 1.0	3. jun 2008
programmer 	hugo
tested by		tobias

FT_PIW is a PI controller.
The PID controller works according to the fomula Y = IN *(KP+ KI * INTEG(e) ).
a rst will reset the integrator to 0
ilim_h and iLim_l set the possible output range of the internal integrator.
the output flag lim will signal that the output limits are active.
the controller is equipped with anti wind_up circuitry that stops the integrator when lim_h or lim_l is reached


default values for KP = 1, KI = 1, ILIM_L = -1E37, iLIM_H = +1E38.
*)

(* run integrator *)
integ(IN := IN, K := KI, RUN := NOT LIM, RST := RST);

(* set output value *)
Y := KP * IN + integ.Out;

(* check for limits and set integrator for anti wind up *)
IF Y < LIM_L THEN
	Y := LIM_L;
	LIM := TRUE;
ELSIF Y > LIM_H THEN
	Y := LIM_H;
	LIM := TRUE;
ELSE
	LIM := FALSE;
END_IF;



(* revision history
hm 	3. jun. 2008 	rev 1.0
	original version


*)

END_FUNCTION_BLOCK

// POUs/Engineering/automation/FT_Profile
FUNCTION_BLOCK FT_Profile
VAR_INPUT
	K : REAL := 1.0;
	O : REAL;
	M : REAL := 1.0;
	E : BOOL;
END_VAR
VAR_INPUT CONSTANT
	value_0 : REAL;
	time_1 : TIME;
	value_1 : REAL;
	time_2 : TIME;
	value_2 : REAL;
	time_3 : TIME;
	value_3 : REAL;
	time_10 : TIME;
	value_10 : REAL;
	time_11 : TIME;
	value_11 : REAL;
	time_12 : TIME;
	value_12 : REAL;
	time_13 : TIME;
	value_13 : REAL;
END_VAR
VAR_OUTPUT
	Y : REAL;
	RUN : BOOL;
	ET : TIME;
END_VAR
VAR
	tx : TIME;
	edge : BOOL;
	state: BYTE;
	ta: TIME;
	tb: TIME;
	t0 : TIME;
	temp: REAL;
	va: REAL;
	vb: REAL;
END_VAR

(*
version 1.1	15 sep 2007
programmer 	tobias
tested by		hugo

FT_Profile generates an output signal which is defined by values over a time scale.
the different values are connected by ramps between the individual values.
a rising edge on E starts the output signal generation and E = True can delay time_3 / value_3 as long as it stays true.
an additional multiplier K can be used to multiply the output and an offset O can be added to the output dynamically.
*)

(* read system time *)
tx := DWORD_TO_TIME(T_PLC_MS());

(* determine start condition *)
IF E AND NOT edge THEN
	RUN := TRUE;
	ET := t#0s;
	t0 := tx;
	ta := tx;
	tb := multime(time_1, M);
	va := value_0;
	vb := value_1;
	temp := value_0;
	state := 1;
END_IF;
edge := E;

(* generate startup profile *)
IF run THEN
	CASE state OF
		1:	IF tx - ta >= tb THEN
				ta := ta + tb;
				tb := multime(time_2 - time_1, M);
				va := value_1;
				vb := value_2;
				temp := value_1;
				state := 2;
			ELSE
				temp := ((vb - va) * TIME_TO_REAL(tx - ta) / TIME_TO_REAL(tb) + va);
			END_IF;
		2:	IF tx - ta >= tb THEN
				ta := ta + tb;
				tb := multime(time_3 - time_2, M);
				va := value_2;
				vb := value_3;
				temp := value_2;
				state := 3;
			ELSE
				temp := ((vb - va) * TIME_TO_REAL(tx - ta) / TIME_TO_REAL(tb) + va);
			END_IF;
		3:	IF tx - ta >= tb THEN
				ta := ta + tb;
				tb := multime(time_10 - time_3, M);
				va := value_3;
				vb := value_10;
				temp := value_3;
				state := 4;
			ELSE
				temp := ((vb - va) * TIME_TO_REAL(tx - ta) / TIME_TO_REAL(tb) + va);
			END_IF;
		4 :	IF tx - ta >= tb THEN
				ta := ta + tb;
				tb := multime(time_11 - time_10, M);
				va := value_10;
				vb := value_11;
				temp := value_10;
				IF E THEN state := 5; ELSE state := 6; END_IF;
			ELSE
				temp := ((vb - va) * TIME_TO_REAL(tx - ta) / TIME_TO_REAL(tb) + va);
			END_IF;
		5:	(* extend the signal while E is true *)
			IF E THEN
				ta := tx;
			ELSE
				state := 6;
			END_IF;
		6:	IF tx - ta >= tb THEN
				ta := ta + tb;
				tb := multime(time_12 - time_11, M);
				va := value_11;
				vb := value_12;
				temp := value_11;
				state := 7;
			ELSE
				temp := ((vb - va) * TIME_TO_REAL(tx - ta) / TIME_TO_REAL(tb) + va);
			END_IF;
		7:	IF tx - ta >= tb THEN
				ta := ta + tb;
				tb := multime(time_13 - time_12, M);
				va := value_12;
				vb := value_13;
				temp := value_12;
				state := 8;
			ELSE
				temp := ((vb - va) * TIME_TO_REAL(tx - ta) / TIME_TO_REAL(tb) + va);
			END_IF;
		8:	IF tx - ta >= tb THEN
				temp := value_13;
				run := FALSE;
			ELSE
				temp := ((vb - va) * TIME_TO_REAL(tx - ta) / TIME_TO_REAL(tb) + va);
			END_IF;
	END_CASE;
	Y := temp * K + O;
	ET := tx - t0;
END_IF;

(* revision history
hm	27 feb 2007		rev 1.0
	original version

hm	15. sep2007		rev 1.1
	replaced Time() with T_PLC_MS for compatibility and performance reasons

*)

END_FUNCTION_BLOCK

// POUs/Engineering/control/FT_PT2
FUNCTION_BLOCK FT_PT2
VAR_INPUT
	in : REAL;
	T : TIME;
	D : REAL;
	K : REAL := 1.0;
END_VAR
VAR_OUTPUT
	out : REAL;
END_VAR
VAR
	init: BOOL;
	int1 : INTEGRATE;
	int2 : INTEGRATE;
	tn: REAL;
	I1, I2 : REAL;
	tn2: REAL;
END_VAR

(*
version 1.5	11. mar. 2009
programmer 	hugo
tested by		oscat

FT_PT2 is a 2nd grade filter with programmable times T, D and faktor K.
 
*)

(* startup initialisation *)
IF NOT init OR T = T#0s THEN
	init := TRUE;
	out := K * in;
	I2 := out;
ELSE
	TN := TIME_TO_REAL(T) * 1.0E-3;
	tn2 := TN * TN;
	int1(X := in * K / tn2 - I1 * 0.5 * D / TN - I2 / TN2, Y := I1);
	int2(X := I1,Y := I2);
	out := I2;
END_IF;


(* revision history

15.1.2007 hm		rev 1.1
	changed formula to new more acurate formula

hm 15.9.2007		rev 1.2
	deleted unused code for init system time reading tx	

hm	30.11.2007	rev 1.3
	changed out to be K * in during initialization
	avoind divide by 0 if tn = 0

hm	3. nov. 2008	rev 1.4
	optimized code and fixed a problem with init

hm	11. mar. 2009	rev 1.5
	real constants updated to new systax using dot

*)

END_FUNCTION_BLOCK

// POUs/Mathematical/functions/FT_RMP
FUNCTION_BLOCK FT_RMP
VAR_INPUT
	Rmp : BOOL := TRUE;
	in : REAL;
	KR : REAL;
	KF : REAL;
END_VAR
VAR_OUTPUT
	out : REAL;
	busy : BOOL;
	UD : BOOL;
END_VAR
VAR
	tx: TIME;
	last: TIME;
	init: BOOL;
END_VAR

(*
	version 1.4	25 jan 2008
	programmer 	oscat
	tested BY		oscat

this ramp function follows an input signal with a linear ramp up or down, the up or down speed can be set with KF and KR.
a K factor of 1 means 1 unit per second on the output. K factors can only be positive and not negative.
a busy output signals the ramp is running or busy false means the in value is present on the output.
a rmp input false means the output follows the input dierctly while a rmp = true means the output follows the input with a ramp.
a updn output signal the directon of the ramp (up or down).

*)

(* read system time *)
tx := DWORD_TO_TIME(T_PLC_MS()) - last;

IF NOT init THEN
	init := TRUE;
	last := tx;
	tx := t#0s;
	out := in;
END_IF;
IF NOT rmp THEN
	out := in;
	busy := FALSE;
ELSIF out > in THEN
	(* ramp down *)
	out := out - TIME_TO_REAL(tx) * 0.001 * KF;
	out := MAX(in, out);
ELSIF out < in THEN
	(* ramp up *)
	out := out + TIME_TO_REAL(tx) * 0.001 * KR;
	out := MIN(in, out);
END_IF;

(* set busy and dir flags *)
IF out < in THEN
	busy := TRUE;
	ud := TRUE;
ELSIF out > in THEN
	busy := TRUE;
	ud := FALSE;
ELSE
	busy := FALSE;
END_IF;
last := last + tx;


(* revision history:

hm 8.10.2006			rev 1.1
	added ud output

hm 12. feb 2007		rev 1.2
	added init variable and corrected a possible startup problem

hm	17. sep 2007	rev 1.3
	replaced time() with t_plc_ms() for compatibility reasons

hm	25. jan 2008	rev 1.4
	performance improvements
	allow KR and KF to be 0
*)

END_FUNCTION_BLOCK

// POUs/Engineering/control/FT_TN16
FUNCTION_BLOCK FT_TN16
VAR_INPUT
	in : REAL;
	T : TIME;
END_VAR
VAR_OUTPUT
	out : REAL;
	trig : BOOL;
END_VAR
VAR
	length : INT := 16;
	X : ARRAY[0..15] OF REAL;
	cnt : INT;
	last : TIME;
	tx: TIME;
	init: BOOL;
END_VAR

(*
version 1.1	16 sep 2007
programmer 	hugo
tested by		tobias

FT_TN16 is delay function, it will delay a signal by a specified time : T and will store 16 values of in before they are put thru to out.
for higher or lower resolution please use FT_TN8 or FT_TN64 instead.
 
*)

(* read system time *)
tx := DWORD_TO_TIME(T_PLC_MS());

trig := FALSE;
IF NOT init THEN
	x[cnt] := in;
	init := TRUE;
	last := tx;
ELSIF tx - last >= T / length THEN
	IF cnt = length - 1 THEN cnt := 0; ELSE cnt := cnt + 1; END_IF;
	Out := X[cnt];
	x[cnt] := in;
	last := tx;
	Trig := TRUE;
END_IF;

(* revision history
hm		1. jan 2007	rev 1.0
	original version

hm		16. sep 2007	rev 1.1
	changes time() to T_plc_ms() for compatibility reasons

*)

END_FUNCTION_BLOCK

// POUs/Engineering/control/FT_TN8
FUNCTION_BLOCK FT_TN8
VAR_INPUT
	in : REAL;
	T : TIME;
END_VAR
VAR_OUTPUT
	out : REAL;
	trig: BOOL;
END_VAR
VAR
	length : INT := 8;
	X : ARRAY[0..7] OF REAL;
	cnt : INT;
	last : TIME;
	tx: TIME;
	init: BOOL;
END_VAR

(*
version 1.1	15 Sep 2007
programmer 	hugo
tested by		tobias

FT_TN8 is delay function, it will delay a signal by a specified time : T and will store 8 values of in before they are put thru to out.
if higher resolution is needed, pls use FT_TN16 or FT_TN64 instead.
 
*)

tx := DWORD_TO_TIME(T_PLC_MS());
trig := FALSE;
IF NOT init THEN
	x[cnt] := in;
	init := TRUE;
	last := tx;
ELSIF tx - last >= T / length THEN
	IF cnt = length - 1 THEN cnt := 0; ELSE cnt := cnt + 1; END_IF;
	Out := X[cnt];
	x[cnt] := in;
	last := tx;
	trig := TRUE;
END_IF;

(* revision history
hm		1. jan 2007		rev 1.0
	original version

hm		16. sep 2007	rev 1.1
	changes time() to T_plc_ms() for compatibility reasons

*)

END_FUNCTION_BLOCK

// POUs/Engineering/control/FT_TN64
FUNCTION_BLOCK FT_TN64
VAR_INPUT
	in : REAL;
	T : TIME;
END_VAR
VAR_OUTPUT
	out : REAL;
	trig: BOOL;
END_VAR
VAR
	length : INT := 64;
	X : ARRAY[0..63] OF REAL;
	cnt : INT;
	last : TIME;
	tx: TIME;
	init: BOOL;
END_VAR

(*
version 1.1	15 sep 2007
programmer 	hugo
tested by		tobias

FT_TN7 is delay function, it will delay a signal by a specified time : T and will store 64 values of in before they are put thru to out.
if lower resolution is needed, pls use FT_TN8 or FT_TN16 instead.
 
*)

(* read system time *)
tx := DWORD_TO_TIME(T_PLC_MS());

trig := FALSE;
IF NOT init THEN
	x[cnt] := in;
	init := TRUE;
	last := tx;
ELSIF tx - last >= T / length THEN
	IF cnt = length - 1 THEN cnt := 0; ELSE cnt := cnt + 1; END_IF;
	Out := X[cnt];
	x[cnt] := in;
	last := tx;
	trig := TRUE;
END_IF;

(* revision history
hm		1. jan 2007		rev 1.0
	original version

hm		16. sep 2007	rev 1.1
	changes time() to T_plc_ms() for compatibility reasons

*)

END_FUNCTION_BLOCK

// POUs/Mathematical/GAUSS
FUNCTION GAUSS : REAL
VAR_INPUT
	X : REAL;
	U : REAL;
	SI: REAL;
END_VAR
VAR
	temp: REAL;
	si_inv: REAL;
END_VAR


(*
version 1.2	10. mar. 2009
programmer 	hugo
tested by		tobias

this function calculates the gaussian density function

*)

temp := X - U;
si_inv := 1.0  / si;
GAUSS := EXP(Temp * Temp * si_inv * si_inv * - 0.5) * 0.39894228 * si_inv;



(* revision hisdtory
hm	6. apr. 2008	rev 1.0
	original version

hm	27. oct. 2008	rev 1.1
	optimized performance	

hm	10. mar. 2009	rev 1.2
	real constants updated to new systax using dot

*)

END_FUNCTION

// POUs/Mathematical/GAUSSCD
FUNCTION GAUSSCD : REAL
VAR_INPUT
	X : REAL;
	U : REAL;
	SI: REAL;
END_VAR


(*
version 1.1	10. mar. 2009
programmer 	hugo
tested by		tobias

this function calculates the gaussian cumulative distribution function

*)

GAUSSCD := (ERF((X - U) / (SI * 1.414213562)) + 1.0) * 0.5;



(* revision hisdtory
hm	6. apr. 2008	rev 1.0
	original version

hm	10. mar. 2009	rev 1.1
	real constants updated to new systax using dot

*)

END_FUNCTION

// POUs/Mathematical/GCD
FUNCTION GCD : INT
VAR_INPUT
	A : DINT;
	B : DINT;
END_VAR
VAR
	t: DINT;
END_VAR


(*
version 1.0	19. jan. 2011
programmer 	hugo
tested by	tobias

this function calculates the gretaest common divisor of two numbers A and B

*)

IF A = 0 THEN
	GCD := DINT_TO_INT(ABS(B));
ELSIF B = 0 THEN
	GCD := DINT_TO_INT(ABS(A));
ELSE
	A := ABS(A);
	B := ABS(B);
	GCD := 1;
	WHILE NOT(A.0 OR B.0) DO
		A := SHR(A,1);
		B := SHR(B,1);
		GCD := SHL(GCD,1);
	END_WHILE;
	WHILE A > 0 DO
		IF NOT(A.0) THEN A := SHR(A,1);
		ELSIF NOT(B.0) THEN B := SHR(B,1);
		ELSE
			t:= SHR(ABS(A-B),1);
			IF A < B THEN B := t; ELSE A := T; END_IF;
		END_IF;
	END_WHILE;
	GCD := GCD * DINT_TO_INT(B);
END_IF;


(* revision history
hm	19. jan. 2011	rev 1.0
	original version

*)

END_FUNCTION

// POUs/Mathematical/GDF
FUNCTION GDF : REAL
VAR_INPUT
	X : REAL;
END_VAR


(*
version 1.2	10. mar. 2009
programmer 	hugo
tested by		tobias

this function calculates the Gudermannian function.

*)

IF X = 0.0 THEN
	GDF := 0.0;
ELSIF X > 15.0 THEN
	GDF := math.PI05;
ELSIF X < -15.0 THEN
	GDF := -math.PI05;
ELSE
	GDF := ATAN(EXP(X)) * 2.0 - math.PI05;
END_IF;

(* revision history
hm	27. apr. 2008	rev 1.0
	original version

hm	18. oct. 2008	rev 1.1
	using math constants

hm	10. mar. 2009	rev 1.2
	real constants updated to new systax using dot

*)

END_FUNCTION

// POUs/Logic/generators/GEN_BIT
FUNCTION_BLOCK GEN_BIT
VAR_INPUT
	in0 : DWORD;
	in1 : DWORD;
	in2 : DWORD;
	in3 : DWORD;
	clk : BOOL;
	steps : INT;
	rep : INT;
	rst : BOOL;
END_VAR
VAR_OUTPUT
	Q0 :BOOL;
	Q1 :BOOL;
	Q2 :BOOL;
	Q3 :BOOL;
	cnt : INT;
	run : BOOL;
END_VAR
VAR
	r0: DWORD;
	r1: DWORD;
	r2: DWORD;
	r3: DWORD;
	rx : INT := 1;
END_VAR

(*
version 1.2	14. mar. 2009
programmer 	hugo
tested by		tobias

gen_bit is 4 bit sequencial pattern generator with 4 DWORD inputs and 4 serial outputs.
with the first clock pulse after a reset or after power on, bit 0 of the input DWORDS IN is present on the Outputs Q and the next clock cycle shifts to Bit 1 and so on.
the input steps defines how many bits of the input dwords will be shifted to the outputs. the sequence can be repetive when rep = 0 or any amount of repetitions can be defined with input rep.

*)

(* check if number of runs is finished or rep = 0 which means continuous *)

IF clk AND NOT rst THEN
	run := (rep = 0) OR (rx <= rep);
	IF run THEN
		(* check for step counter reached and reset to 0 if cnt = steps *)
		IF cnt = steps THEN
			cnt := 0;
		END_IF;

		(* when cnt = 0 then reload the inputs into the registers *)
		IF cnt = 0 THEN
			r0 := in0;
			r1 := in1;
			r2 := in2;
			r3 := in3;
		END_IF;

		(* when cnt < steps, shift the lowest bits to the outputs *)
		IF (cnt < steps) THEN
			Q0 := r0.0;
			Q1 := r1.0;
			Q2 := r2.0;
			Q3 := r3.0;
			r0 := SHR(r0,1);
			r1 := SHR(r1,1);
			r2 := SHR(r2,1);
			r3 := SHR(r3,1);
		END_IF;

		(* increment the step counter *)
		cnt := cnt +1;
		IF (cnt = steps) AND (rep <> 0) THEN rx := rx +1; END_IF;
		IF (rx > rep) AND (rep <> 0) THEN run := FALSE; END_IF;
	END_IF;
ELSE
	IF rst THEN
		run := FALSE;
		Q0 := FALSE;
		Q1 := FALSE;
		Q2 := FALSE;
		Q3 := FALSE;
		r0 := 0;
		r1 := 0;
		r2 := 0;
		r3 := 0;
		cnt := 0;
		rx := 1;
	END_IF;
END_IF;



(* revision histroy
hm	4 aug 2006	rev 1.0
	original version

hm 15. oct. 2008	rev 1.1
	improved performance

hm	14. mar. 2009	rev 1.2
	removed double assignments

*)

END_FUNCTION_BLOCK

// POUs/Engineering/signal generators/GEN_PULSE
FUNCTION_BLOCK GEN_PULSE
VAR_INPUT
	ENQ : BOOL := TRUE;
	PTH : TIME;
	PTL : TIME;
END_VAR
VAR_OUTPUT
	Q : BOOL;
END_VAR
VAR
	tx: TIME;
	tn: TIME;
	init: BOOL;
END_VAR

(*
version 1.5	8. apr. 2011
programmer 	hugo
tested by		oscat

GEN_PULSE uses the internal sps timer to generate a continuous output waveform with programmable high and low time.
the accuracy of gen_pulse is depending on the system timer.
when time is 0 the high and low times are exactly one cycle.
ENQ = TRUE will start and ENQ = FALSE will stop the generator.

*)

IF enq THEN
	tx := DWORD_TO_TIME(T_PLC_MS());
	IF NOT init THEN init := TRUE; tn := tx; END_IF;
	IF tx - tn >= SEL(Q, PTL, PTH) THEN
		tn := tn + SEL(Q, PTL, PTH);
		Q := NOT Q;
	END_IF;
ELSE
	Q := FALSE;
	init := FALSE;
END_IF;



(* revision history
hm	29. jun. 2008	rev 1.0
	original version

hm	23. nov. 2008	rev 1.1
	set default for enq to be true

hm	18. jul. 2009	rev 1.2
	improved performance

hm	13. nov. 2009	rev 1.3
	corrected error

hm	16. feb. 2011	rev 1.4
	corrected an error when timer overflows

hm	8. apr. 2011	rev 1.5
	ptl and pth was exchanged
*)

END_FUNCTION_BLOCK

// POUs/Engineering/signal generators/GEN_PW2
FUNCTION_BLOCK GEN_PW2
VAR_INPUT
	ENQ : BOOL;
	TH1 : TIME;
	TL1 : TIME;
	TH2 : TIME;
	TL2 : TIME;
	TS : BOOL;
END_VAR
VAR_OUTPUT
	Q : BOOL;
	TH : TIME;
	TL : TIME;
END_VAR
VAR
	t_high : TIME;
	t_low : TIME;
	tx : TIME;
	start : TIME;
	init : BOOL;
	et : TIME;
END_VAR

(*
version 1.1	14. mar. 2009
programmer 	hugo
tested by		oscat

GEN_PW2 generates a time TH? followed by a time TL?.
the input ts selects between 2 sets of timings for the operation.


*)

(* read system timer *)
tx := DWORD_TO_TIME(T_PLC_MS());

(* startup initialization *)
IF NOT init THEN
	start := tx;
	init := TRUE;
	TH := T#0s;
	TL := T#0s;
END_IF;

(* timing selection *)
IF TS THEN
	t_high := TH2;
	t_low := TL2;
ELSE
	t_high := TH1;
	t_low := TL1;
END_IF;

(* normal operation *)
IF ENQ THEN
	et := tx - start;
	IF NOT Q THEN
		IF et >= t_low THEN
			Q := TRUE;
			start := tx;
			TL := T#0s;
		ELSE
			TL := et;
		END_IF;
	ELSE
		IF et >= t_high THEN
			Q := FALSE;
			start := tx;
			TH := T#0s;
		ELSE
			TH := et;
		END_IF;
	END_IF;
ELSE
	Q := FALSE;
	TH := T#0s;
	TL := T#0s;
	start := tx;
END_IF;



(* revision history
hm	26. sep. 2008	rev 1.0
	original version

hm	14. mar. 2009	rev 1.1
	removed double assignments

*)

END_FUNCTION_BLOCK

// POUs/Engineering/signal generators/GEN_RDM
FUNCTION_BLOCK GEN_RDM
VAR_INPUT
	PT : TIME;
	AM : REAL := 1;
	OS : REAL;
END_VAR
VAR_OUTPUT
	Q : BOOL;
	Out : REAL;
END_VAR
VAR
	tx : TIME;
	last : TIME;
	init : BOOL;
END_VAR

(*
	version 1.1	16 sep 2007
	programmer 	oscat
	tested BY		oscat

this signal generator generates a random output. The signal is defined by period time (PT), 
amplitude (AM), offset (OS).
The Output waveform will have its max peak at AM/2 + OS and its minimum peak at -AM/2 + OS. 
The period time PT defines how often the output signal will jump to a new randow value.
The Output Q will be true for one cycle anytime the output OUT has changed

*)

(* read system time and prepare input data *)
tx := DWORD_TO_TIME(T_PLC_MS()) - last;

(* init section *)
IF NOT init THEN
	init := TRUE;
	last := tx;
	tx := t#0s;
END_IF;

(* add last if one cycle is finished *)
IF tx >= pt THEN
	last := last + pt;
	tx := tx - pt;

	(* generate output signal *)
	out := am * (RDM(0) - 0.5) + os;
	q := TRUE;
ELSE
	q := FALSE;
END_IF;

(* revision history

hm	7.2.2007		rev 1.0
	original version

hm	16.9.2007		rev 1.1
	changes time() to T_plc_ms() for compatibility reasons

*)

END_FUNCTION_BLOCK

// POUs/Engineering/signal generators/GEN_RDT
FUNCTION_BLOCK GEN_RDT

VAR_INPUT
	Enable		 : BOOL := TRUE ;
	Min_Time_ms	: TIME := t#1s ; (* min Taktzeit *)
	Max_Time_ms	: TIME := t#1.2s ; (* Max Taktzeit *)
	TP_Q		 : TIME := t#100ms ; (* Zeit Ausgang auf TRUE *)
END_VAR
VAR_OUTPUT
	xQ		 : BOOL ;
END_VAR
VAR
	(* Taktgenerator Simulation *)
	tonRDMTimer	: TON ; (* Zeitbaustein Taktgenerator *)
	tof_xQ		: TOF ; (* Ausschaltverzögerung Taktgenerator *)
	tRDMTime	: TIME ; (* Sollzeit *)
	rRDMTime	: REAL ; (* Zufalswert Timer *)
END_VAR

(*
version 1.1	16 mar. 2008
programmer 	J. Schohaus
tested by		Hugo

RDMT generates a defined pulse with pulse width TP_Q at random times. the random time will be defined with an minimum and maximum time.

*)


(*
FUNCTION_BLOCK RDMTimer
###############################################################################
		 Ersteller / author :		 		 		 		 		 J.Schohaus
		 Datum / date:		 		 		 		 		 		 13.07.2007
###############################################################################
		 Änderungen / Datum / Ersteller :		 		 		 		 		 		 		 		 		 		 		 		 		 		 		 
		 moditication / date / author :		 		 
###############################################################################
		 Verwendete Bibliotheken		 ( * werden im Baustein nicht benötigt )
		 		 		 		 Oscat.lib
###############################################################################
Beschreibung:
*)

tonRDMTimer ( IN:= Enable , PT:= tRDMTime );
tof_xQ ( IN:= tonRDMTimer.Q , PT:= TP_Q );
XQ := tof_xq.Q;
IF tonRDMTimer.Q THEN
		 xQ := TRUE ;
		 rRDMTime := RDM ( last:= rRDMTime ) ;
		 tRDMTime := REAL_TO_TIME ( rRDMTime * DINT_TO_REAL(TIME_TO_DINT( Max_Time_ms - Min_Time_ms ) + TIME_TO_DINT(Min_Time_ms ))) ;
		 tonRDMTimer ( IN:= FALSE );
END_IF;

(* revision history
J. Schohaus	19. nov 2007	rev 1.0
	origial version

hm	16. mar. 2008			rev 1.1
	added type conversion to avoid warnings under codesys 3.0
*)

END_FUNCTION_BLOCK

// POUs/Engineering/signal generators/GEN_RMP
FUNCTION_BLOCK GEN_RMP
VAR_INPUT
	PT : TIME := t#1s;
	AM : REAL := 1.0;
	OS : REAL;
	DL : REAL;
END_VAR
VAR_OUTPUT
	Q : BOOL;
	OUT : REAL;
END_VAR
VAR
	tx : TIME;
	last : TIME;
	init : BOOL;
	temp : REAL;
	ltemp: REAL;
END_VAR

(*
	version 1.4	10. mar. 2009
	programmer 	oscat
	tested BY		oscat

this signal generator generates a ramp wave output. The ramp wave signal is defined by period time (PT), 
amplitude (AM), offset (OS) and a specific delay for the output signal (DL).
The Output waveform will have its minimum peak at OS and its maximum peak at AM + OS. 
The delay input can delay a signal up to PT, this can be useful to synchronize different generators 
and generate interleaving signals.
in addition to the analog output Out there is a second boolean output Q with is true for one cycle when the ramp starts.
*)

(* read system time and prepare input data *)
tx := DWORD_TO_TIME(T_PLC_MS()) - last;
DL := MODR(dl,1.0);
IF dl < 0.0 THEN dl := 1.0 - dl; END_IF;

(* init section *)
IF NOT init THEN
	init := TRUE;
	last := tx;
	tx := t#0s;
END_IF;

(* add last if one cycle is finished *)
IF tx >= pt THEN
	last := last + pt;
	tx := tx - pt;
END_IF;

(* generate sine wave *)
ltemp := temp;
IF pt > t#0s THEN temp := FRACT(TIME_TO_REAL(tx + MULTIME(pt, dl)) / TIME_TO_REAL(pt)); END_IF;
out := am * temp + os;

(* boolean output Q *)
Q := temp < ltemp;

(* revision history
hm	3. mar 2007		rev 1.0
	original version

hm	17 sep 2007		rev 1.1
	replaced time() with t_plc_ms for compatibilitx reasons

hm	27. nov 2007	rev 1.2
	avoid divide by 0 when pt = 0

ks	26. oct. 2008	rev 1.3
	code optimization

hm	10. mar. 2009	rev 1.4
	changed real constants to use dot syntax
*)

END_FUNCTION_BLOCK

// POUs/Engineering/signal generators/GEN_SIN
FUNCTION_BLOCK GEN_SIN
VAR_INPUT
	PT : TIME;
	AM : REAL := 1.0;
	OS : REAL;
	DL : REAL;
END_VAR
VAR_OUTPUT
	Q : BOOL;
	Out : REAL;
END_VAR
VAR
	tx : TIME;
	last : TIME;
	init : BOOL;
	temp : REAL;
END_VAR

(*
version 1.6	11. mar. 2009
programmer 	oscat
tested BY	oscat

this signal generator generates a sine wave output. The sine wave signal is defined by period time (PT), 
amplitude (AM), offset (OS) and a specific delay for the output signal (DL).
The Output waveform will have its max peak at AM/2 + OS and its minimum peak at -AM/2 + OS. 
The delay input can delay a signal up to PT, this can be useful to synchronize different generators 
and generate interleaving signals. A Cos wave can be generated accordingly.
in addition to a analog output Out there is a second boolean output Q with the corresponding binary signal.
*)

(* read system time and prepare input data *)
tx := DWORD_TO_TIME(T_PLC_MS()) - last;
DL := MODR(dl,1.0);
IF dl < 0.0 THEN dl := 1.0 - dl; END_IF;

(* init section *)
IF NOT init THEN
	init := TRUE;
	last := tx;
	tx := t#0s;
END_IF;

(* add last if one cycle is finished *)
IF tx >= pt THEN
	last := last + pt;
	tx := tx - pt;
END_IF;

(* generate sine wave *)
IF pt > t#0s THEN temp := SIN(math.PI2 * DWORD_TO_REAL(TIME_TO_DWORD(tx + MULTIME(pt, dl))) / DWORD_TO_REAL(TIME_TO_DWORD(pt))); END_IF;
out := am * 0.5 *  temp + os;

(* boolean output Q *)
q := NOT SIGN_R(temp);

(* revision history
hm	22. jan 2007	rev 1.0
	original version

hm	17 sep 2007	rev 1.1
	replaced time() with t_plc_ms for compatibilitx reasons

hm	27. nov 2007	rev 1.2
	avoid divide by 0 when pt = 0

hm	6. jan 2008		rev 1.3
	improved performance

hm	16. mar. 2008	rev 1.4
	added type conversion to avoid warnings under codesys 3.0

hm	18. oct. 2008	rev 1.5
	using math constants

hm	11. mar. 2009	rev 1.6
	changed real constants to use dot syntax

*)

END_FUNCTION_BLOCK

// POUs/Logic/generators/GEN_SQ
FUNCTION_BLOCK GEN_SQ
VAR_INPUT
	PT : TIME;
END_VAR
VAR_OUTPUT
	Q : BOOL;
END_VAR
VAR
	tn: DWORD;
	tx: DWORD;
	init : BOOL;
END_VAR

(*
version 1.3	16. feb. 2011
programmer 	hugo
tested by		tobias

gen_sq generates square wave signal with programmable period time.

*)

(* read system time *)
tx := T_PLC_MS();

IF NOT init THEN
	init := TRUE;
	tn := tx;
	Q := TRUE;
ELSIF tx - tn >= SHR(TIME_TO_DWORD(PT),1) THEN
	Q := NOT Q;
	tn := tn + SHR(TIME_TO_DWORD(pt),1);
END_IF;


(* revision history
hm	4. aug 2006	rev 1.0
	original version

hm	17. sep 2007	rev 1.1
	replaced time() with T_PLC_MS() for compatibility reasons

hm	18. jul. 2009	rev 1.2
	improved accuracy

hm	16. feb 2011	rev 1.3
	corrected an error with timer overflow 
*)

END_FUNCTION_BLOCK

// POUs/Engineering/signal generators/GEN_SQR
FUNCTION_BLOCK GEN_SQR
VAR_INPUT
	PT : TIME;
	AM : REAL := 1.0;
	OS : REAL;
	DC : REAL := 0.5;
	DL : REAL;
END_VAR
VAR_OUTPUT
	Q : BOOL;
	Out : REAL;
END_VAR
VAR
	tx : TIME;
	last : TIME;
	init: BOOL;
END_VAR

(*
version 1.4	11. mar. 2009
programmer 	oscat
tested BY		oscat

this signal generator generates a square wave output. The square wave signal is defined by period time (PT), 
amplitude (AM), offset (OS), duty cycle (DC) and a specific delay for the output signal (DL).
The Output waveform will switch between AM/2 + OS and -AM/2 + OS. The DC input specifies ther duty cycle, 
DC = 0 means output is low at all times and 1 means output is high at all times.
The delay input can delay a signal up to PT, this can be useful to synchronize different generators and generate interleaving signals.
in addition to a analog output Out there is a second boolean output Q.
*)

(* check dc = 1 or 0 *)
IF dc = 0.0 THEN
	out := -am * 0.5 + os;
	Q := FALSE;
	RETURN;
ELSIF dc = 1.0 THEN
	out := am * 0.5 + os;
	Q := TRUE;
	RETURN;
END_IF;

(* read system time and prepare input data *)
tx := DWORD_TO_TIME(T_PLC_MS()) - last;
DL := MODR(dl,1.0);
IF dl < 0.0 THEN dl := 1.0 - dl; END_IF;
dc := MODR(dc,1.0);
IF dc < 0.0 THEN dc := 1.0 - dc; END_IF;

(* init section *)
IF NOT init THEN
	init := TRUE;
	last := tx;
	tx := t#0s;
END_IF;

(* add last if one cycle is finished *)
IF tx >= pt THEN
	last := last + pt;
	tx := tx - pt;
END_IF;

(* check if falling or rising edge first *)
IF MULTIME(pt, dl + dc) >= pt THEN
	(* generate falling edge *)
	IF tx >= MULTIME(pt, dl + dc - 1) THEN
		out := -am * 0.5 + os;
		Q := FALSE;
	END_IF;
	(* generate rising edge *)
	IF tx >= MULTIME(pt, dl) THEN
		out := am * 0.5 + os;
		Q := TRUE;
	END_IF;
ELSE
	(* generate rising edge first *)
	IF tx >= MULTIME(pt, dl) THEN
		out := am * 0.5 + os;
		Q := TRUE;
	END_IF;
	(* generate falling edge *)
	IF tx >= MULTIME(pt, dl + dc) THEN
		out := -am * 0.5 +os;
		Q := FALSE;
	END_IF;
END_IF;

(* revision history

hm	12. feb 2007	rev 1.1
	added default value for dc = 0.5

hm	17 sep 2007	rev 1.2
	replaced time() with t_plc_ms for compatibilitx reasons

hm	6. jan 2008	rev 1.3
	improved performance

hm	11. mar. 2009	rev 1.4
	changed real constants to use dot syntax
	set default amplitude to 1.0

*)

END_FUNCTION_BLOCK

// POUs/Engineering/conversion/GEO_TO_DEG
FUNCTION GEO_TO_DEG : REAL
VAR_INPUT
	D : INT;
	M : INT;
	SEC : REAL;
END_VAR


(*
version 1.0	22. jan. 2009
programmer 	hugo
tested by		oscat

this function converts degrees, minutes seconds to decimal degrees.

*)

GEO_TO_DEG := INT_TO_REAL(D) + INT_TO_REAL(M) * 0.016666666666667 + sec * 0.00027777777777778;


(* revision histroy
hm	22. jan. 2009	rev 1.0
	original release


*)

END_FUNCTION

// POUs/Mathematical/GOLD
FUNCTION GOLD : REAL
VAR_INPUT
	X : REAL;
END_VAR


(*
version 1.1	10. mar. 2009
programmer 	hugo
tested by		tobias

this function calculates the golden function.

*)

GOLD := (X + SQRT(X*X + 4.0)) * 0.5;


(* revision history
hm	27. apr. 2008	rev 1.0
	original version

hm	10. mar. 2009	rev 1.1
	real constants updated to new systax using dot

*)

END_FUNCTION

// POUs/Logic/gate logic/GRAY_TO_BYTE
FUNCTION GRAY_TO_BYTE : BYTE
VAR_INPUT
	IN : BYTE;
END_VAR


(*
version 1.0	9. nov. 2009
programmer 	hugo
tested by		oscat

this function converts a gray code into binary

*)

GRAY_TO_BYTE := SHR(IN,4) XOR IN;
GRAY_TO_BYTE := SHR(GRAY_TO_BYTE,2) XOR GRAY_TO_BYTE;
GRAY_TO_BYTE := SHR(GRAY_TO_BYTE,1) XOR GRAY_TO_BYTE;

(* revision history
hm	9. nov. 2009	rev 1.0
	original version

*)

END_FUNCTION

// POUs/Time&Date/HOUR_OF_DT
FUNCTION HOUR_OF_DT : INT
VAR_INPUT
	XDT : DT;
END_VAR


(*
	version 1.0	6. jun. 2008
	programmer 	oscat
	tested BY	oscat

HOUR_OF_DT returns the current hour (hour of the day) of a DT variable

*)

HOUR_OF_DT := DWORD_TO_INT((DT_TO_DWORD(XDT) MOD 86400) / 3600);


(* revision history
hm		6.9.2008	rev 1.0
	original version


*)

END_FUNCTION

// POUs/Engineering/control/HYST
FUNCTION_BLOCK HYST
VAR_INPUT
	In : REAL;
	ON : REAL;
	OFF : REAL;
END_VAR
VAR_OUTPUT
	Q : BOOL;
	win : BOOL;
END_VAR


(*
version 1.0	2. jun. 2008
programmer 	hugo
tested BY	oscat

This Hystereses function has two modes:
1. if on > off then Q will be switched high when in > on and switched low when in < off.
2. if on < off then Q will be switched high when in < on and switched low when in > off.
the output win will be high when in is between low and high.

*)

IF ON >= OFF THEN
	IF IN < OFF THEN
		Q := FALSE;
		WIN := FALSE;
	ELSIF  IN > ON THEN
		Q := TRUE;
		WIN := FALSE;
	ELSE
		WIN := TRUE;
	END_IF;
ELSE
	IF IN > OFF THEN
		Q := FALSE;
		WIN := FALSE;
	ELSIF  IN < ON THEN
		Q := TRUE;
		WIN := FALSE;
	ELSE
		WIN := TRUE;
	END_IF;
END_IF;


(* revision history
hm		2.  jun 2008	rev 1.0
	original version

*)

END_FUNCTION_BLOCK

// POUs/Engineering/control/HYST_1
FUNCTION_BLOCK HYST_1
VAR_INPUT
	In : REAL;
	high : REAL;
	low : REAL;
END_VAR
VAR_OUTPUT
	Q : BOOL;
	win : BOOL;
END_VAR


(*
version 1.1	2. jun. 2008
programmer 	hugo
tested BY	oscat

this hysteresis function switches the output high if the input signal reaches obove high and will switch to low when the input falls back below low value.
a separate output mid is set if the input stays between low and high value.

*)

IF in < low THEN
	Q := FALSE;
	win := FALSE;
ELSIF in > high THEN
	Q := TRUE;
	win := FALSE;
ELSE
	win := TRUE;
END_IF;




(* revision history
hm		4.  aug. 2006	rev 1.0
	original version

hm		2. jun. 2008	rev 1.1
	improved performance
*)

END_FUNCTION_BLOCK

// POUs/Engineering/control/HYST_2
FUNCTION_BLOCK HYST_2
VAR_INPUT
	IN : REAL;
	VAL : REAL;
	HYS : REAL;
END_VAR
VAR_OUTPUT
	Q : BOOL;
	WIN: BOOL;
END_VAR
VAR
	tmp: REAL;
END_VAR


(*
version 1.2	2. jun. 2008
programmer 	oscat
tested BY	oscat

this hysteresis function switches the output high if the input signal reaches obove val + hys/2 and will switch to low when the input falls back below val - hys/2 value.
a separate output mid is set if the input stays between low and high value.

*)

tmp := val - hys * 0.5;
IF in < tmp THEN
	Q := FALSE;
	win := FALSE;
ELSIF in > tmp + hys THEN
	Q := TRUE;
	win := FALSE;
ELSE
	win := TRUE;
END_IF;



(* revision history
hm		4. aug 2006	rev 1.0
	original version

hm		5. jan 2008	rev 1.1
	improved code for better performance

hm		2. jun. 2008	rev 1.2
	improved performance
*)

END_FUNCTION_BLOCK

// POUs/Engineering/control/HYST_3
FUNCTION_BLOCK HYST_3
VAR_INPUT
	in : REAL;
	hyst : REAL;
	val1 : REAL;
	val2 : REAL;
END_VAR
VAR_OUTPUT
	Q1 : BOOL;
	Q2 : BOOL;
END_VAR
VAR
	X: REAL;
END_VAR

(*
version 1.2	5 jan 2008
programmer 	oscat
tested BY	oscat

this is a double hysteresis function. Out1 follows a hysteresis function defined by val1and hyst, while out 2 follows val2 and hyst.
if the input signal is between the two hysteresis switches (val1 and val2) then non of the outputs is active.

*)

X := hyst * 0.5;
IF in < val1 - X THEN
	q1 := TRUE;
ELSIF in > val1 + X THEN
	q1 := FALSE;
END_IF;
IF in < val2 - X THEN
	q2 := FALSE;
ELSIF in > val2 + X THEN
	q2 := TRUE;
END_IF;



(* revision history
hm	22. jan 2007	rev 1.0
	original version

hm	27. dec 2007	rev 1.1
	changed code for better performance

hm	5. jan 2008	rev 1.2
	further performance iprovements

*)

END_FUNCTION_BLOCK

// POUs/Mathematical/INC2
FUNCTION INC2 : INT
VAR_INPUT
	X : INT;
	D : INT;
	L : INT;
	U : INT;
END_VAR
VAR
	tmp: INT;
END_VAR


(*
version 1.0	29. jun. 2008
programmer 	hugo
tested by	oscat

This function increments the input X by the value D and compares the result with U.
if the output exceeds U it will continue to count from L again.

*)

tmp := U - L + 1;
INC2 := (X + D - L + tmp) MOD tmp + L;



(* revision history
hm	29. jun. 2008		REV 1.0
	original version


*)

END_FUNCTION

// POUs/Engineering/automation/INC_DEC
FUNCTION_BLOCK INC_DEC
VAR_INPUT
	CHa : BOOL;
	CHb : BOOL;
	RST : BOOL;
END_VAR
VAR_OUTPUT
	dir : BOOL;
	cnt : INT;
END_VAR
VAR
	edgea : BOOL;
	clk: BOOL;
	clka: BOOL;
	clkb: BOOL;
	edgeb: BOOL;
	axb: BOOL;
END_VAR

(*
	version 1.0	4 aug 2006
	programmer 	oscat
	tested BY		oscat

incremental decoder with quadruple accuracy.
2 pulses for each channel are created for each directional pulse.
*)

axb := cha XOR chb;

(* create pulses for channel a *)
clka := cha XOR edgea;
edgea := cha;

clkb := chb XOR edgeb;
edgeb := chb;

(* create pulses for both channels *)
clk := clka OR clkb;

(* set the direction output *)
IF axb AND clka THEN dir := TRUE; END_IF;
IF axb AND clkb THEN dir := FALSE; END_IF;

(* increment or decrement the counter *)
IF clk AND dir THEN cnt := cnt + 1; END_IF;
IF clk AND NOT dir THEN cnt := cnt -1; END_IF;

(* reset the counter if rst active *)
IF rst THEN cnt := 0; END_IF;

END_FUNCTION_BLOCK

// POUs/Logic/gate logic/INT_TO_BCDC
FUNCTION INT_TO_BCDC : BYTE
VAR_INPUT
	IN : INT;
END_VAR


(*
version 1.1	30. jun. 2008
programmer 	hugo
tested by		tobias

this function converts an integer into a two digit bcd number.
*)

INT_TO_BCDC := SHL(INT_TO_BYTE(IN / INT#10),4) OR INT_TO_BYTE(in MOD INT#10);

(* revision history
hm	13.12.2007
	original version

hm	30.6.2008	rev 1.1
	changed name INT_TO_BCD to INT_TO_BCDC to avoid collision with util.lib
	corrected error in code

*)

END_FUNCTION

// POUs/Engineering/automation/INTERLOCK
FUNCTION_BLOCK INTERLOCK
VAR_INPUT
	I1, I2 : BOOL;
	TL : TIME;
END_VAR
VAR_OUTPUT
	Q1, Q2 : BOOL;
END_VAR
VAR
	T1, T2 : TOF;
END_VAR

(*
version 1.0	28 sep 2007
programmer 	hugo
tested by		tobias

INTERLOCK has two inputs I1 and I2 which drive the corresponding outputs Q1 and Q2.
the inputs signals lock each other out and therfore I1 can only drive Q1 when I2 is Low and vice versa.
The input TL specifies a dead time between two outputs can become active.
an output can only become active when the other output was not active for the time TL.

*)

(* the input signal have a run delay to lockout the other input *)
T1(IN := I1, PT := TL);
T2(IN := I2, PT := TL);

Q1 := I1 AND NOT t2.Q;
Q2 := I2 AND NOT t1.Q;


(* revision history

hm	28 sep 2007		rev 1.0
	original version

*)

END_FUNCTION_BLOCK

// POUs/Engineering/automation/INTERLOCK_4
FUNCTION_BLOCK INTERLOCK_4
VAR_INPUT CONSTANT
END_VAR
VAR_INPUT
	I0 : BOOL;
	I1 : BOOL;
	I2 : BOOL;
	I3 : BOOL;
	E : BOOL;
	MODE : INT;

END_VAR
VAR_OUTPUT
	OUT : BYTE;
	TP : BOOL;
END_VAR
VAR
	in: BYTE;
	last: BYTE;
	old: BYTE;
	lmode: INT;
END_VAR

(*
version 1.1	14. mar. 2009
programmer 	hugo
tested by		oscat

INTERLOCK_4 detects one of 4 switches and delivers the number of the switch pressed on the output out
a output tp is true for one cycle if the output has changed.
a setup variable MODE selects between 3 different modes:
MODE = 0, any input active will disable all other inputs
MODE = 1, the input with the highest number will be acepted
mode = 2, the input last pressed will disable all others 

*)

(* check if enable is active *)
IF E THEN
(* reset all vars when there is a mode change on thy fly *)
	IF mode <> lmode THEN
		out := 0;
		last := 0;
		old := 0;
		lmode := mode;
	END_IF;
	(* load inputs into in *)
	in.0 := I0;
	in.1 := I1;
	in.2 := I2;
	in.3 := I3;
	(* only execute when there is any change *)
	IF in <> last THEN
		(* only execute when inputs have chages state *)
		CASE mode OF
			0:	(* output directly display inputs as bits in byte out *)
				out := in;

			1:	(* the input with the highest number will be acepted *)
				IF in.3 THEN out := 8;
				ELSIF in.2 THEN out := 4;
				ELSIF in.1 THEN out := 2;
				ELSE out := in;
				END_IF;

			2:	(* input last pressed will be displayed only *)
				last := ((in XOR last) AND in);
				IF last.3 THEN out := 8;
				ELSIF last.2 THEN out := 4;
				ELSIF last.1 THEN out := 2;
				ELSE out := last;
				END_IF;

			3:	(* any input active will disable all other inputs *)
				IF (out AND in) = 0 THEN
					IF in.3 THEN out := 8;
					ELSIF in.2 THEN out := 4;
					ELSIF in.1 THEN out := 2;
					ELSE out := in;
					END_IF;
				END_IF;

		END_CASE;
		last := in;
	END_IF;
	tp := out <> old;
	old := out;
ELSE
	out := 0;
	last := 0;
	old := 0;
	lmode := 0;
	tp := FALSE;
END_IF;


(* revision history
hm	24. oct 2008	rev 1.0
	original version

hm	14. mar. 2009	rev 1.1
	replaced double assignments

*)

END_FUNCTION_BLOCK

// POUs/String/IS_ALNUM
FUNCTION IS_ALNUM : BOOL
VAR_INPUT
	str : STRING(STRING_LENGTH);
END_VAR
VAR
	L: INT;
	pt : POINTER TO BYTE;
	pos: INT;
END_VAR

(*
version 1.1	29. mar. 2008
programmer 		kurt
tested by		hugo

ISC_ALNUM testet ob in einem string nur Zahlen 0..9 vorkommen.

*)

PT := ADR(str);
L := LEN(str);
FOR pos := 1 TO L DO
	IF NOT (ISC_ALPHA(pt^) OR ISC_NUM(pt^)) THEN
		IS_ALNUM := FALSE;
		RETURN;
	END_IF;
    	PT := PT + 1;
END_FOR;
IS_ALNUM := L > 0;


(* revision history
hm	29. feb 2008	rev 1.0
	original version

hm	29. mar. 2008	rev 1.1
	changed STRING to STRING(STRING_LENGTH)
*)

END_FUNCTION

// POUs/String/ISC_ALPHA
FUNCTION ISC_ALPHA : BOOL
VAR_INPUT
	IN : BYTE;
END_VAR


(*
version 1.1	19. oct. 2008
programmer 	oscat
tested by	oscat

ISC_ALPHA checks if a character is a..z or A..Z.

*)

IF setup.EXTENDED_ASCII THEN
	ISC_ALPHA := (in > 64 AND in < 91) OR (in > 191  AND in <> 215 AND in <> 247) OR (in > 96 AND in < 123);
ELSE
	ISC_ALPHA := (IN > 64 AND IN < 91) OR (in > 96 AND in < 123);
END_IF;

(* revision history
hm	6. mar. 2008	rev 1.0
	original version

hm	19. oct. 2008	rev 1.1
	changes setup constants
*)

END_FUNCTION

// POUs/String/ISC_NUM
FUNCTION ISC_NUM : BOOL
VAR_INPUT
	IN : BYTE;
END_VAR


(*
version 1.0	6. mar 2008
programmer 	oscat
tested by		hugo

ISC_NUM checks if a character is 0..9.

*)

ISC_NUM := IN > 47 AND IN < 58;

(* revision history
hm		6. mar. 2008	rev 1.0
	original version

*)

END_FUNCTION

// POUs/String/IS_ALPHA
FUNCTION IS_ALPHA : BOOL
VAR_INPUT
	str : STRING(STRING_LENGTH);
END_VAR
VAR
	L: INT;
	pt : POINTER TO BYTE;
	pos: INT;
END_VAR

(*
version 1.1	29. mar. 2008
programmer 		kurt
tested by		hugo

IS_ALPHA testet ob in einem string nur Zeichen a-z oder A - Z vorkommen.

*)

PT := ADR(str);
L := LEN(str);
FOR pos := 1 TO L DO
	IF NOT ISC_ALPHA(pt^) THEN
		IS_ALPHA := FALSE;
		RETURN;
	END_IF;
    	PT := PT + 1;
END_FOR;
IS_ALPHA := L > 0;


(* revision history
hm	29. feb 2008	rev 1.0
	original version

hm	29. mar. 2008	rev 1.1
	changed STRING to STRING(STRING_LENGTH)
*)

END_FUNCTION

// POUs/String/IS_CC
FUNCTION IS_CC : BOOL
VAR_INPUT
	str : STRING(STRING_LENGTH);
	cmp : STRING(STRING_LENGTH);
END_VAR
VAR
	L: INT;
	pos: INT;
END_VAR

(*
version 1.1	29. mar. 2008
programmer 	Tobias
tested by	hugo

ISC_CC testet ob ein string nur aus Zeichen des Strings CMP besteht.

*)

L := LEN(str);
FOR pos := 1 TO L DO
	IF FIND(CMP,MID(str,1,pos)) = 0 THEN RETURN; END_IF;
END_FOR;
IS_CC := L > 0;



(* revision history
hm	19. mar 2008	rev 1.0
	original version

hm	29. mar. 2008	rev 1.1
	changed STRING to STRING(STRING_LENGTH)
*)

END_FUNCTION

// POUs/String/IS_CTRL
FUNCTION IS_CTRL : BOOL
VAR_INPUT
	STR : STRING(STRING_LENGTH);
END_VAR
VAR
	L: INT;
	pt : POINTER TO BYTE;
	pos: INT;
END_VAR

(*
version 1.1	29. mar 2008
programmer 		kurt
tested by		hugo

IS_CTRL testet ob in einem string nur Steuerzeichen (Char < 32) vorkommen.

*)

PT := ADR(str);
L := LEN(str);
FOR pos := 1 TO L DO
	IF NOT (ISC_CTRL(pt^)) THEN
		IS_CTRL := FALSE;
		RETURN;
	END_IF;
    	PT := PT + 1;
END_FOR;
IS_CTRL := L > 0;


(* revision history
hm	29. feb. 2008	rev 1.0
	original version

hm	29. mar. 2008	rev 1.1
	changed STRING to STRING(STRING_LENGTH)
*)

END_FUNCTION

// POUs/String/ISC_CTRL
FUNCTION ISC_CTRL : BOOL
VAR_INPUT
	IN : BYTE;
END_VAR


(*
version 1.0	6. mar 2008
programmer 	oscat
tested by		hugo

ISC_ALPHA checks if a character is a control character.

*)

ISC_CTRL := IN < 32 OR IN = 127;

(* revision history
hm		6. mar. 2008	rev 1.0
	original version

*)

END_FUNCTION

// POUs/String/IS_HEX
FUNCTION IS_HEX : BOOL
VAR_INPUT
	str : STRING(STRING_LENGTH);
END_VAR
VAR
	L: INT;
	pt : POINTER TO BYTE;
	pos: INT;
END_VAR

(*
version 1.1	29. mar. 2008
programmer 		kurt
tested by		hugo

IS_HEX testet ob in einem string nur Zahlen 0..9 oder A..F oder a..f  vorkommen.

*)

PT := ADR(str);
L := LEN(str);
FOR pos := 1 TO L DO
	IF NOT (ISC_HEX(pt^)) THEN
		IS_HEX := FALSE;
		RETURN;
	END_IF;
    	PT := PT + 1;
END_FOR;
IS_HEX := L > 0;


(* revision history
hm	29. feb 2008	rev 1.0
	original version

hm	29. mar. 2008	rev 1.1
	changed STRING to STRING(STRING_LENGTH)
*)

END_FUNCTION

// POUs/String/ISC_HEX
FUNCTION ISC_HEX : BOOL
VAR_INPUT
	IN : BYTE;
END_VAR


(*
version 1.0	6. mar 2008
programmer 	oscat
tested by		hugo

ISC_HEX checks if a character is 0..9, A..F, a..f.

*)

ISC_HEX := (IN > 47 AND IN < 58) OR (IN > 64 AND IN < 71) OR (IN > 96 AND IN < 103);

(* revision history
hm		6. mar. 2008	rev 1.0
	original version

*)

END_FUNCTION

// POUs/String/IS_LOWER
FUNCTION IS_LOWER : BOOL
VAR_INPUT
	str : STRING(STRING_LENGTH);
END_VAR
VAR
	l: INT;
	pt : POINTER TO BYTE;
	pos: INT;
END_VAR

(*
version 1.1	29. mar. 2008
programmer 		kurt
tested by		hugo

IS_LOWER testet ob in einem string nur kleinbuchstaben vorkommen.

*)

PT := ADR(str);
L := LEN(str);
FOR pos := 1 TO L DO
	IF NOT (ISC_LOWER(pt^)) THEN
		IS_LOWER := FALSE;
		RETURN;
	END_IF;
    	PT := PT + 1;
END_FOR;
IS_LOWER := L > 0;


(* revision history
hm	29. feb 2008	rev 1.0
	original version

hm	29. mar. 2008	rev 1.1
	changed STRING to STRING(STRING_LENGTH)
*)

END_FUNCTION

// POUs/String/ISC_LOWER
FUNCTION ISC_LOWER : BOOL
VAR_INPUT
	IN : BYTE;
END_VAR


(*
version 1.1	19. oct. 2008
programmer 	hugo
tested by	oscat

isc_lower checks if a character is lowercase.

*)

IF setup.EXTENDED_ASCII THEN
	ISC_LOWER := ((in > 96) AND (in < 123)) OR ((in > 222) AND (in <> 247));
ELSE
	ISC_LOWER := ((in > 96) AND (in < 123));
END_IF;

(* revision history
hm	6. mar. 2008	rev 1.0
	original version

hm	19. oct. 2008	rev 1.1
	changes setup constants
*)

END_FUNCTION

// POUs/String/IS_NCC
FUNCTION IS_NCC : BOOL
VAR_INPUT
	str : STRING(STRING_LENGTH);
	cmp : STRING(STRING_LENGTH);
END_VAR
VAR
	L: INT;
	pos: INT;
END_VAR

(*
version 1.1	29. mar. 2008
programmer 	Tobias
tested by		hugo

IS_NCC testet ob in einem string keine Zeichen des Strings CMP enthalten sind.

*)

L := LEN(str);
FOR pos := 1 TO L DO
	IF FIND(CMP,MID(str,1,pos)) > 0 THEN RETURN; END_IF;
END_FOR;
IS_NCC := TRUE;



(* revision history
hm	19. mar 2008	rev 1.0
	original version

hm	29. mar. 2008	rev 1.1
	changed STRING to STRING(STRING_LENGTH)
*)

END_FUNCTION

// POUs/String/IS_NUM
FUNCTION IS_NUM : BOOL
VAR_INPUT
	str : STRING(STRING_LENGTH);
END_VAR
VAR
	L : INT;
	pt : POINTER TO BYTE;
	pos: INT;
END_VAR

(*
version 1.1	29. mar. 2008
programmer 		kurt
tested by		hugo

IS_NUM testet ob in einem string nur Zahlen 0..9 vorkommen.

*)

PT := ADR(str);
L := LEN(str);
FOR pos := 1 TO L DO
	IF NOT (ISC_NUM(pt^)) THEN
		IS_NUM := FALSE;
		RETURN;
	END_IF;
    	PT := PT + 1;
END_FOR;
IS_NUM := L > 0;


(* revision history
hm	29. feb 2008	rev 1.0
	original version

hm	29. mar. 2008	rev 1.1
	changed STRING to STRING(STRING_LENGTH)
*)

END_FUNCTION

// POUs/Mathematical/Array/IS_SORTED
FUNCTION IS_SORTED : BOOL
VAR_INPUT
	pt : POINTER TO ARRAY[0..32000] OF REAL;
	size : UINT;
END_VAR
VAR

	stop: INT;
	i: INT;
END_VAR

(*
version 1.1	4. apr. 2008
programmer 	hugo
tested by	tobias

this function will return true if the given array is sorted in an ascending order.
the function needs to be called:	array_sorted(adr("array"),sizeof("array"));
because this function works with pointers its very time efficient and it needs no extra memory.

*)

stop := UINT_TO_INT(SHR(size,2)-2);
FOR i := 0 TO stop DO
	IF pt^[i] > pt^[i+1] THEN
		IS_SORTED := FALSE;
		RETURN;
	END_IF;
END_FOR;

IS_SORTED := TRUE;

(* revision history

hm 	29. mar. 2008 	rev 1.0
	original version

hm	4. apr. 2008	rev 1.1
	added type conversion to avoid warnings under codesys 3.0
*)

END_FUNCTION

// POUs/String/IS_UPPER
FUNCTION IS_UPPER : BOOL
VAR_INPUT
	str : STRING(STRING_LENGTH);
END_VAR
VAR
	L: INT;
	pt : POINTER TO BYTE;
	pos: INT;
END_VAR

(*
version 1.1	29. mar. 2008
programmer 		kurt
tested by		hugo

IS_UPPER testet ob in einem string keine Kleinbuchstaben vorkommen.

*)

PT := ADR(str);
L := LEN(str);
FOR pos := 1 TO L DO
	IF NOT (ISC_UPPER(pt^)) THEN
		IS_UPPER := FALSE;
		RETURN;
	END_IF;
    	PT := PT + 1;
END_FOR;
IS_UPPER := L > 0;


(* revision history
hm	29. feb 2008	rev 1.0
	original version

hm	29. mar. 2008	rev 1.1
	changed STRING to STRING(STRING_LENGTH)
*)

END_FUNCTION

// POUs/String/ISC_UPPER
FUNCTION ISC_UPPER : BOOL
VAR_INPUT
	IN : BYTE;
END_VAR


(*
version 1.1	19. oct. 2008
programmer 	hugo
tested by	oscat

ISC_upper checks if a character is uppercase

*)

IF setup.EXTENDED_ASCII THEN
	ISC_UPPER :=  ((in > 64) AND (in < 91)) OR (((in > 191) AND (in < 223)) AND (in <> 215));
ELSE
	ISC_UPPER := ((in > 64) AND (in < 91));
END_IF;


(* revision history
hm	6. mar. 2008	rev 1.0
	original version

hm	19. oct. 2008	rev 1.1
	changes setup constants

*)

END_FUNCTION

// POUs/Time&Date/JD2000
FUNCTION JD2000 : REAL
VAR_INPUT
	DTI : DT;
END_VAR


(*
version 1.0	15. jul. 2008
programmer 	hugo
tested by	oscat

JULIAN calculates the astronomic julian date from 1.1.2000-12:00.

*)

JD2000 := DWORD_TO_REAL(DT_TO_DWORD(DTI) - 946728000) / 86400.0;

(* revision histroy
hm	15. jul. 2008	rev 1.0
	original release


*)

END_FUNCTION

// POUs/Engineering/conversion/K_TO_C
FUNCTION K_TO_C : REAL
VAR_INPUT
	Kelvin : REAL;
END_VAR


(*
version 1.1	19. aug 2009
programmer 	hugo
tested by		tobias

this function converts kelvin to celsius

*)

K_TO_C := Kelvin + phys.T0;


(* revision history

hm	4. aug 2006	rev 1.0
	original version

hm	19. aug 2009	rev 1.1
	fixed calculation error

*)

END_FUNCTION

// POUs/Engineering/conversion/KMH_TO_MS
FUNCTION KMH_TO_MS : REAL
VAR_INPUT
	kmh : REAL;
END_VAR


(*
version 1.1	6 jan 2007
programmer 	hugo
tested by		tobias

this function converts velocities from Kilometers / hour to Meters / Second

*)

KMH_TO_MS := kmh * 0.2777777777777;

(* revision history
hm	4. feb 2007		rev 1.0
	original version

hm	6. jan 2008		rev 1.1
	improved performance

*)

END_FUNCTION

// POUs/Mathematical/LAMBERT_W
FUNCTION LAMBERT_W : REAL
VAR_INPUT
	X : REAL;
END_VAR
VAR
	w : REAL;
	i : INT;
	we: REAL;
	w1e: REAL;
	last: DWORD;
	ewx: REAL;
END_VAR



(*
version 1.1	10. mar. 2009
programmer 	hugo
tested by		oscat

this function calculates the lambert_w function.

*)

(* check for valid input and return -1000 if too low *)
IF x < -0.367879441171442 THEN
	LAMBERT_W := -1000.0;
	RETURN;
(* return 0 if x = 0 *)
ELSIF x = 0.0 THEN
	RETURN;
(* first an estimate is calculated *)
ELSIF x <= 500.0 THEN
	w := LN(x + 1.0);
	w := 0.665 * (1.0 + 0.0195 * w) * w + 0.04;
ELSE
	w := LN(x - 4.0) - (1.0 - 1.0/LN(x)) * LN(LN(x));
END_IF;
(* use estimate to calculate exact result *)
FOR i := 0 TO 5 DO
	ewx := EXP(w);
	we := w * ewx - x;
	w1e := (w+1.0) * ewx;
	last := REAL_TO_DW(w) AND 16#FFFF_FFFC;
	w := w - (we / (w1e - (w+2.0) * we / (2.0 * w + 2.0)));
	IF (REAL_TO_DW(w) AND 16#FFFF_FFFC) = last THEN EXIT; END_IF;
END_FOR;
LAMBERT_W := w;


(* revision hisdtory
hm	26. oct. 2008	rev 1.0
	original version

hm	10. mar. 2009	rev 1.1
	real constants updated to new systax using dot

*)

END_FUNCTION

// POUs/Logic/gate logic/REAL_TO_DW
FUNCTION REAL_TO_DW : DWORD
VAR_INPUT
	X : REAL;
END_VAR
VAR
	pt : POINTER TO DWORD;
END_VAR

(*
version 1.0	18. apr. 2008
programmer 	hugo
tested by		tobias

this function converts a 32 Bit Real to a dword in a bitwise manner.
*)

pt := ADR(X);
REAL_TO_DW := pt^;

(* revision history
hm	18. apr. 2008
	original version

*)

END_FUNCTION

// POUs/Mathematical/LANGEVIN
FUNCTION LANGEVIN : REAL
VAR_INPUT
	X : REAL;
END_VAR


(*
version 1.2	10.mar. 2009
programmer 	hugo
tested by		tobias

